			IF (GVL.A_RunStep <= GVL.A_LengthStep)
			   AND F_IsMotionCmd(
					GVL_1.Step_Cr_A[GVL.A_RunStep].Cmd
			   )
			THEN
	
				//----------------------------------------
				// Đồng bộ step tiếp theo cần Push
				//----------------------------------------
// 				GVL.A_PipelineNextPushStep :=
// 					GVL.A_RunStep;
				GVL.A_RunState := 100;
				IF (GVL.A_RunMode = 1) THEN
					GVL.A_StepHold := TRUE;
				END_IF;
				
	
			ELSE
	
				// Gặp END_WHILE hoặc logic khác
				GVL.A_RunState := 130;
	
			END_IF;
	
		END_IF;
		



    130: // WAIT ALL MOTION CLEAR BEFORE LOGIC

		//--------------------------------------------------------
		// Chờ queue và toàn bộ slot motion thực sự sạch
		//--------------------------------------------------------
		IF (GVL.A_MotionCount <= 0)
		   AND (GVL.A_ActiveMotionCount <= 0)
		   AND NOT GVL.A_MotionManagerBusy
		THEN
			//----------------------------------------------------
			// Reset trạng thái phiên pipeline vừa kết thúc
			//----------------------------------------------------
			GVL.A_PipelineActive := FALSE;
// 			GVL.A_PipelineNextPushStep := 0;
// 	
// 			GVL.A_PushMotionReq := FALSE;
// 			GVL.A_PushMotionDone := FALSE;
// 			GVL.A_PushMotionError := FALSE;
// 	
// 			//----------------------------------------------------
// 			// Xóa phản hồi completion của chuỗi motion vừa chạy
// 			//----------------------------------------------------
// 			GVL.A_MotionDonePulse := FALSE;
// 			GVL.A_MotionDoneStep := 0;
// 	
// 			GVL.A_MotionErrorPulse := FALSE;
// 			GVL.A_MotionErrorStep := 0;
// 			GVL.A_MotionErrorCode := 0;
	
			//----------------------------------------------------
			// Quay lại READ STEP để chạy lệnh logic:
			// END_WHILE, IF, WAIT, END...
			//----------------------------------------------------
			GVL.A_RunState := 0;
		END_IF;
		
	140: // WAIT MOTION CLEAR BEFORE WHILE RESTART

		//--------------------------------------------------------
		// Chờ toàn bộ motion của vòng hiện tại hoàn thành
		//--------------------------------------------------------
		IF (GVL.A_MotionCount <= 0)
		   AND (GVL.A_ActiveMotionCount <= 0)
		   AND NOT GVL.A_MotionManagerBusy
		THEN
			//----------------------------------------------------
			// Hạ request của pipeline
			//----------------------------------------------------
			GVL.A_PushMotionReq := FALSE;
			GVL.A_PipelineActive := FALSE;
	
			//----------------------------------------------------
			// Sang bước reset handshake
			//----------------------------------------------------
			MotionCycleResetScan := 0;
			GVL.A_RunState := 141;
		END_IF;
		
	141: // RESET MOTION PIPELINE BEFORE NEXT WHILE LOOP

		CASE MotionCycleResetScan OF
	
			0:
				//------------------------------------------------
				// Scan thứ nhất: xóa các tín hiệu phiên cũ
				//------------------------------------------------
				GVL.A_PushMotionReq := FALSE;
				GVL.A_PushMotionDone := FALSE;
				GVL.A_PushMotionError := FALSE;
	
				GVL.A_PipelineActive := FALSE;
				GVL.A_PipelineNextPushStep := 0;
	
				GVL.A_MotionDonePulse := FALSE;
				GVL.A_MotionDoneStep := 0;
	
				GVL.A_MotionErrorPulse := FALSE;
				GVL.A_MotionErrorStep := 0;
				GVL.A_MotionErrorCode := 0;
	
				MotionCycleResetScan := 1;
	
	
			1:
				//------------------------------------------------
				// Scan thứ hai:
				// fbPushMotion đã được gọi với Execute=FALSE.
				// Motion FB đã được gọi với Start=FALSE.
				//------------------------------------------------
				IF NOT GVL.A_PushMotionReq
				   AND (GVL.A_MotionCount <= 0)
				   AND (GVL.A_ActiveMotionCount <= 0)
				   AND NOT GVL.A_MotionManagerBusy
				THEN
					MotionCycleResetScan := 0;
	
					//--------------------------------------------
					// Bây giờ mới quay lại WHILE
					//--------------------------------------------
					GVL.A_RunStep := WhileReturnStep;
					GVL.A_RunState := 0;
				END_IF;
	
		END_CASE;
	
    900: // ERROR
        GVL.A_RunBusy := FALSE;
        GVL.A_PushMotionReq := FALSE;
        GVL.A_PipelineActive := FALSE;

END_CASE;


//====================================================
// FB Push Motion Queue phải gọi mỗi scan
//====================================================
fbPushMotion(
    Execute := GVL.A_PushMotionReq,
    Item := GVL.A_PushMotionItem
);

GVL.A_PushMotionDone  := fbPushMotion.Done;
GVL.A_PushMotionError := fbPushMotion.Error;
END_ACTION

ACTION PRG_A_MotionManager:
//====================================================
// PRG_A_MotionManager
// Controlled Pipeline Motion Manager
// - Chạy nền liên tục.
// - Có queue và slot rảnh thì Pop motion vào slot.
// - Slot Accepted thì hạ Start để FB Motion chạy tiếp.
// - Slot Done thì báo về Interpreter bằng A_MotionDonePulse.
// - Slot Error thì báo lỗi đúng SourceStep.
//====================================================


//====================================================
// ABORT REQUEST
// Ưu tiên cao nhất trong MotionManager
// Dùng khi Stop / Alarm / Reset
//====================================================
IF GVL.A_MotionAbortReq OR GVL.X[7] THEN

    PopReq := FALSE;

    GVL.A_MotionHead := 1;
    GVL.A_MotionTail := 1;
    GVL.A_MotionCount := 0;
	GVL.A_PipelineUsedCount := 0;
    FOR i := 1 TO 3 DO
        GVL.A_MoveSlotStart[i] := FALSE;
        GVL.A_MoveSlotBusy[i] := FALSE;

        GVL.A_MoveSlotAccepted[i] := FALSE;
        GVL.A_MoveSlotDone[i] := FALSE;
        GVL.A_MoveSlotError[i] := FALSE;
        GVL.A_MoveSlotErrorID[i] := 0;
		GVL.A_MoveSlotReleasePending[i] := FALSE;
        GVL.A_MoveSlotCmd[i] := E_RobotCmd.CMD_NOP;
		
    END_FOR;

    GVL.A_ActiveMotionCount := 0;

    GVL.A_MotionManagerBusy := FALSE;
    GVL.A_MotionManagerDone := FALSE;
    GVL.A_MotionManagerError := FALSE;
    GVL.A_MotionManagerState := 0;

    GVL.A_MotionDonePulse := FALSE;
    GVL.A_MotionErrorPulse := FALSE;

    GVL.A_MotionAbortReq := FALSE;
    GVL.A_MotionAbortDone := TRUE;

ELSE

	// Luôn gọi FB MoveP/L/C mỗi scan
	
	CASE GVL.A_MotionManagerState OF
	
		0: // IDLE / READY
	
			GVL.A_MotionManagerDone := FALSE;
	
			// Nếu có motion trong queue và còn slot rảnh thì lấy ra chạy
			IF (GVL.A_MotionCount > 0) AND (F_GetFreeMoveSlot() > 0) THEN
				GVL.A_MotionManagerBusy := TRUE;
				PopReq := TRUE;
	
				GVL.A_MotionManagerState := 10;
	
			ELSE
				// Không còn queue và không còn slot active
				IF GVL.A_ActiveMotionCount <= 0 THEN
					GVL.A_MotionManagerBusy := FALSE;
				END_IF;
			END_IF;
	
	
		10: // WAIT POP DONE
	
			IF fbPop.Done THEN
				PopReq := FALSE;
	
				item_PRG_A_MotionManager := fbPop.Item;
				freeSlot := F_GetFreeMoveSlot();
	
				IF freeSlot > 0 THEN
	
					// Gán item vào slot rảnh
					GVL.A_MoveSlotItem[freeSlot] := item_PRG_A_MotionManager;
					GVL.A_MoveSlotCmd[freeSlot]  := item_PRG_A_MotionManager.Cmd;
	
					// Reset trạng thái slot trước khi Start
					GVL.A_MoveSlotBusy[freeSlot]     := TRUE;
					GVL.A_MoveSlotStart[freeSlot]    := TRUE;
					GVL.A_MoveSlotAccepted[freeSlot] := FALSE;
					GVL.A_MoveSlotDone[freeSlot]     := FALSE;
					GVL.A_MoveSlotError[freeSlot]    := FALSE;
					
					GVL.A_MoveSlotErrorID[freeSlot] := 0;

					GVL.A_MoveSlotReleasePending[freeSlot] := FALSE;
					
					// Ghi nhớ chính xác slot vừa cấp
   					WaitAcceptSlot := freeSlot;
	
					// Tăng số motion đang active
					//GVL.A_ActiveMotionCount := GVL.A_ActiveMotionCount + 1;
	
					GVL.A_MotionManagerState := 20;
	
				ELSE
					// Trường hợp hiếm: vừa Pop xong nhưng slot không còn rảnh
					GVL.A_MotionManagerState := 30;
				END_IF;
			END_IF;
	
			IF fbPop.Empty THEN
				PopReq := FALSE;
				GVL.A_MotionManagerState := 30;
			END_IF;
	
	
		20: // WAIT COMMAND ACCEPTED
			
		//--------------------------------------------------------
			// Chỉ chờ đúng slot vừa được State 10 cấp lệnh
			//--------------------------------------------------------
			IF (WaitAcceptSlot >= 1)
			   AND (WaitAcceptSlot <= 3)
			THEN
		
				//----------------------------------------------------
				// Slot vẫn phải thuộc quyền sở hữu của Manager
				//----------------------------------------------------
				IF GVL.A_MoveSlotBusy[WaitAcceptSlot] THEN
		
					//------------------------------------------------
					// Lệnh đã được FB Move nhận
					//------------------------------------------------
					IF GVL.A_MoveSlotAccepted[WaitAcceptSlot] THEN
		
						GVL.A_MoveSlotStart[WaitAcceptSlot] := FALSE;
		
						// Đã hoàn thành handshake Accepted
						WaitAcceptSlot := 0;
		
						//--------------------------------------------
						// PipelineLength = 1:
						// Không Pop thêm khi còn motion đang chạy.
						// Sang State 30 chờ motion hoàn thành.
						//--------------------------------------------
						GVL.A_MotionManagerState := 30;
		
		
					ELSIF GVL.A_MoveSlotError[WaitAcceptSlot] THEN
		
						GVL.A_MotionManagerError := TRUE;
		
						GVL.A_MotionErrorPulse := TRUE;
						GVL.A_MotionErrorStep :=
							GVL.A_MoveSlotItem[WaitAcceptSlot].SourceStep;
		
						GVL.A_MotionErrorCode :=
							GVL.A_MoveSlotErrorID[WaitAcceptSlot];
		
						WaitAcceptSlot := 0;
		
						GVL.A_MotionManagerState := 900;
		
					END_IF;
		
				END_IF;
		
			ELSE
		
				//----------------------------------------------------
				// Không có slot nào đang chờ Accepted.
				// Đây là trạng thái bất thường, quay về quản lý queue.
				//----------------------------------------------------
				GVL.A_MotionManagerState := 30;
		
			END_IF;
	
		30: // WAIT / CONTINUE PIPELINE
	
			// Nếu sau đó Interpreter push thêm queue và có slot rảnh thì tiếp tục chạy
			IF (GVL.A_MotionCount > 0) AND (F_GetFreeMoveSlot() > 0) THEN
				GVL.A_MotionManagerBusy := TRUE;
				PopReq := TRUE;
				GVL.A_MotionManagerState := 10;
	
			// Nếu không còn queue và không còn motion active thì MotionManager rảnh
			ELSIF (GVL.A_MotionCount <= 0) AND (GVL.A_ActiveMotionCount <= 0) THEN
				GVL.A_MotionManagerBusy := FALSE;
				GVL.A_MotionManagerDone := TRUE;
				GVL.A_MotionManagerState := 0;
			END_IF;
	
	
		900: // ERROR
	
			PopReq := FALSE;
	
			// Dừng cấp thêm motion mới
			FOR i := 1 TO 3 DO
				GVL.A_MoveSlotStart[i] := FALSE;
			END_FOR;
	
			GVL.A_MotionManagerBusy := FALSE;
			GVL.A_MotionManagerError := TRUE;
	
			GVL.A_MotionManagerState := 0;
	
	END_CASE;
END_IF;
//====================================================
// Gọi FB Pop mỗi scan
//====================================================
fbPop(
    Execute := PopReq
);



//============================================================
// CALL MOTION SLOT FB
// Tất cả FB phải được gọi liên tục mỗi scan.
//
// Khi slot không sử dụng hoặc không đúng loại lệnh:
// Start của FB tương ứng phải bằng FALSE.
// Nhờ vậy LastStart và State bên trong FB được cập nhật đúng.
//============================================================

FOR i := 1 TO 3 DO

    //--------------------------------------------------------
    // Chuẩn bị tọa độ
    //--------------------------------------------------------
    IF GVL.A_MoveSlotBusy[i] THEN

        CASE GVL.A_MoveSlotCmd[i] OF

            E_RobotCmd.CMD_MovP,
            E_RobotCmd.CMD_MovL:

//                 SlotPos[i] :=
//                     F_GetPointSMC_A(
//                         GVL.A_MoveSlotItem[i].PointNo
//                     );
				IF GVL.A_MoveSlotItem[i].UseDirectPosition THEN
					SlotPos[i].c.X := GVL.A_MoveSlotItem[i].DirectPosition.X;
					SlotPos[i].c.Y := GVL.A_MoveSlotItem[i].DirectPosition.Y;
					SlotPos[i].c.Z := GVL.A_MoveSlotItem[i].DirectPosition.Z;
					SlotPos[i].c.A := GVL.A_MoveSlotItem[i].DirectPosition.A;
				ELSE
					SlotPos[i] := F_GetPointSMC_A(GVL.A_MoveSlotItem[i].PointNo);
				END_IF;



            E_RobotCmd.CMD_MovC:

                SlotMidPos[i] :=
                    F_GetPointSMC_A(
                        GVL.A_MoveSlotItem[i].MidPointNo
                    );

                SlotEndPos[i] :=
                    F_GetPointSMC_A(
                        GVL.A_MoveSlotItem[i].EndPointNo
                    );

        END_CASE;

    END_IF;


    //--------------------------------------------------------
    // MoveP
    // Luôn gọi mỗi scan
    //--------------------------------------------------------
    fbMoveP[i](
        Start :=
            GVL.A_MoveSlotBusy[i]
            AND
            (GVL.A_MoveSlotCmd[i] = E_RobotCmd.CMD_MovP)
            AND
            GVL.A_MoveSlotStart[i],
		Release := GVL.A_MoveSlotReleasePending[i],
        AxisGroup := SCARA_A,
        Item := GVL.A_MoveSlotItem[i],
        PositionIn := SlotPos[i],
        //CoordSystem := GVL.RB_A.COORD
		CoordSystem := SEL(
			GVL.A_MoveSlotItem[i].UseDirectPosition,
			//GVL.RB_A.COORD,
			SMC_COORD_SYSTEM.MCS,
			GVL.A_MoveSlotItem[i].DirectCoordSystem)

    );


    //--------------------------------------------------------
    // MoveL
    // Luôn gọi mỗi scan
    //--------------------------------------------------------
    fbMoveL[i](
        Start :=
            GVL.A_MoveSlotBusy[i]
            AND
            (GVL.A_MoveSlotCmd[i] = E_RobotCmd.CMD_MovL)
            AND
            GVL.A_MoveSlotStart[i],

        AxisGroup := SCARA_A,
        Item := GVL.A_MoveSlotItem[i],
        PositionIn := SlotPos[i],
        //CoordSystem := GVL.RB_A.COORD
		CoordSystem := SEL(
			GVL.A_MoveSlotItem[i].UseDirectPosition,
			//GVL.RB_A.COORD,
			SMC_COORD_SYSTEM.MCS,
			GVL.A_MoveSlotItem[i].DirectCoordSystem)

    );


    //--------------------------------------------------------
    // MoveC
    // Luôn gọi mỗi scan
    //--------------------------------------------------------
    fbMoveC[i](
        Start :=
            GVL.A_MoveSlotBusy[i]
            AND
            (GVL.A_MoveSlotCmd[i] = E_RobotCmd.CMD_MovC)
            AND
            GVL.A_MoveSlotStart[i],

        AxisGroup := SCARA_A,
        Item := GVL.A_MoveSlotItem[i],
        MidPosition := SlotMidPos[i],
        EndPosition := SlotEndPos[i],
        //CoordSystem := GVL.RB_A.COORD
		CoordSystem := SMC_COORD_SYSTEM.MCS
    );


	



    //--------------------------------------------------------
    // Chọn trạng thái trả về theo loại lệnh của slot
    //--------------------------------------------------------
    IF GVL.A_MoveSlotBusy[i] THEN

        CASE GVL.A_MoveSlotCmd[i] OF

            //================================================
            // MOVP
            //================================================
            E_RobotCmd.CMD_MovP:

                GVL.A_MoveSlotAccepted[i] :=
                    fbMoveP[i].Accepted;

                GVL.A_MoveSlotDone[i] :=
                    fbMoveP[i].Done;

                GVL.A_MoveSlotError[i] :=
                    fbMoveP[i].Error;

                GVL.A_MoveSlotErrorID[i] :=
                    fbMoveP[i].ErrorID_Custom;


            //================================================
            // MOVL
            //================================================
            E_RobotCmd.CMD_MovL:

                GVL.A_MoveSlotAccepted[i] :=
                    fbMoveL[i].Accepted;

                GVL.A_MoveSlotDone[i] :=
                    fbMoveL[i].Done;

                GVL.A_MoveSlotError[i] :=
                    fbMoveL[i].Error;

                GVL.A_MoveSlotErrorID[i] :=
                    fbMoveL[i].ErrorID_Custom;


            //================================================
            // MOVC
            //================================================
            E_RobotCmd.CMD_MovC:

                GVL.A_MoveSlotAccepted[i] :=
                    fbMoveC[i].Accepted;

                GVL.A_MoveSlotDone[i] :=
                    fbMoveC[i].Done;

                GVL.A_MoveSlotError[i] :=
                    fbMoveC[i].Error;

                GVL.A_MoveSlotErrorID[i] :=
                    fbMoveC[i].ErrorID_Custom;

        END_CASE;

    END_IF;

END_FOR;


//------------------------------------------------------------
// GLOBAL MOTION ERROR MONITOR
//
// Kiểm tra tất cả Move Slot mỗi scan.
// Giữ nguyên cơ chế MotionErrorPulse cũ để báo Interpreter.
//------------------------------------------------------------
IF NOT GVL.A_MotionErrorPulse THEN

    FOR i := 1 TO 3 DO

        IF GVL.A_MoveSlotBusy[i] AND GVL.A_MoveSlotError[i]
        THEN

            //--------------------------------------------
            // MotionManager có lỗi
            //--------------------------------------------
            GVL.A_MotionManagerError := TRUE;

            //--------------------------------------------
            // Xung báo Interpreter
            //--------------------------------------------
            GVL.A_MotionErrorPulse := TRUE;

            //--------------------------------------------
            // Step gây lỗi
            //--------------------------------------------
            GVL.A_MotionErrorStep := GVL.A_MoveSlotItem[i].SourceStep;

            //--------------------------------------------
            // Error Code của FB
            //--------------------------------------------
            GVL.A_MotionErrorCode := GVL.A_MoveSlotErrorID[i];

            //--------------------------------------------
            // Có thể lưu thêm Slot để debug
            //--------------------------------------------
            GVL.A_MotionErrorSlot := i;

            //--------------------------------------------
            // Manager chuyển ERROR
            //--------------------------------------------
            GVL.A_MotionManagerState := 900;

            EXIT;

        END_IF;

    END_FOR;

END_IF;

// RELEASE SLOT WHEN DONE
FOR i := 1 TO 3 DO

    IF GVL.A_MoveSlotBusy[i]
       AND GVL.A_MoveSlotDone[i]
    THEN

        // Báo Interpreter
        GVL.A_MotionDoneStep :=
            GVL.A_MoveSlotItem[i].SourceStep;

        GVL.A_MotionDonePulse := TRUE;

        // Release slot
        GVL.A_MoveSlotStart[i] := FALSE;
        GVL.A_MoveSlotBusy[i] := FALSE;
        GVL.A_MoveSlotAccepted[i] := FALSE;
        GVL.A_MoveSlotDone[i] := FALSE;
        GVL.A_MoveSlotError[i] := FALSE;
        GVL.A_MoveSlotErrorID[i] := 0;

        GVL.A_MoveSlotCmd[i] :=
            E_RobotCmd.CMD_NOP;
		GVL.A_MoveSlotReleasePending[i] := TRUE; // Set release = TRUE
		
		//------------------------------------------------
		// Motion đã thực sự rời pipeline
		//------------------------------------------------
		IF GVL.A_PipelineUsedCount > 0 THEN
			GVL.A_PipelineUsedCount :=
				GVL.A_PipelineUsedCount - 1;
		END_IF;
	
    END_IF;
END_FOR;

//============================================================
// RECALCULATE ACTIVE MOTION COUNT
//
// A_ActiveMotionCount luôn phản ánh đúng số slot Busy,
// không phụ thuộc việc cộng/trừ có bị bỏ sót hay không.
//============================================================
ActiveCountCalc := 0;

FOR i := 1 TO 3 DO

    IF GVL.A_MoveSlotBusy[i] THEN
        ActiveCountCalc := ActiveCountCalc + 1;
    END_IF;

END_FOR;

GVL.A_ActiveMotionCount := ActiveCountCalc;




//====================================================
// FINALIZE MOTION MANAGER
// Chỉ kết thúc khi Manager đã vào trạng thái WAIT
// Không được reset State 10/20 khi vừa Pop lệnh.
//====================================================
IF (GVL.A_MotionManagerState = 30)
   AND (GVL.A_MotionCount <= 0)
   AND (GVL.A_ActiveMotionCount <= 0)
THEN

    GVL.A_MotionManagerBusy := FALSE;
    GVL.A_MotionManagerDone := TRUE;
    GVL.A_MotionManagerState := 0;

END_IF;
END_ACTION

ACTION Main_Base_Program_RB_B:
//=============================================================================
// REPLACE ACTION: Main_Base_Program_RB_B
// SOURCE: current Main_Base_Program_RB_A in PG_MAR_V3_1707_10(4).xml
// METHOD: strict A -> B mirror for robot-specific runtime.
// IMPORTANT: replace the ENTIRE existing Main_Base_Program_RB_B body.
//=============================================================================

//====================================================
// PRG_B_Interpreter
// Controlled Pipeline:
// - Motion được nạp trước tối đa A_PipelineDepth lệnh.
// - A_RunStep chỉ tăng khi step hiện tại Done thật.
// - Gặp lệnh logic thì chờ Motion Queue + Slot sạch.
//====================================================



//====================================================
// STOP COMMAND
//====================================================
IF GVL.B_RunStop OR GVL.X[7] THEN

    // Dừng Interpreter
    GVL.B_RunEnable := FALSE;
    GVL.B_RunBusy := FALSE;
    GVL.B_RunDone := FALSE;
    GVL.B_RunPause := FALSE;
    GVL.B_RunState := 0;
    // GVL.B_RunStop := FALSE;

    // Dừng pipeline
    GVL.B_PipelineActive := FALSE;
    GVL.B_PushMotionReq := FALSE;
    GVL.B_PushMotionDone := FALSE;
    GVL.B_PushMotionError := FALSE;
	// 1707
	//------------------------------------------------
    // Reset bộ nhớ cạnh của FB Push
    //------------------------------------------------
    fbPushMotion_B(
        Execute := FALSE,
        Item := GVL.B_PushMotionItem
    );

    // Yêu cầu MotionManager abort toàn bộ motion pipeline
    GVL.B_MotionAbortReq := TRUE;
	
	// Dừng command Tracking đang chạy.
	IF GVL.B_StepActive THEN
		GVL.g_stMultiTrackCommandB.Abort := TRUE;
		GVL.g_stMultiTrackCommandB.Execute := FALSE;
	
		GVL.B_StepActive := FALSE;
		udiTrackCommandIDB := 0;
	END_IF;
	
	// Hủy Tool command từ Interpreter.
	GVL.g_stInterpreterToolCommandB.Execute := FALSE;
	GVL.g_stInterpreterToolCommandB.Abort := TRUE;
	
	udiToolReleaseCommandIDB := 0;
	// GVL.B_StepActive := FALSE;
	//GVL.g_axDORequestToolB[4] := FALSE;
	
	//xVisionAlignStartB := FALSE;
	// Hủy Vision Request khi Stop/Disable Robot B.

    //=============================================================================
	// ABORT VISION REQUEST - ROBOT B
	//-----------------------------------------------------------------------------
	// Khi Robot Stop, Robot không phát Request mới và hạ Execute hiện tại.
	// Vision Manager sẽ thực hiện phần reset handshake phía Manager.
	//=============================================================================
	GVL.g_stVisionAlignRequestB.Execute := FALSE;
	xVisionStepActiveB := FALSE;

    RETURN;
END_IF;


//====================================================
// NOT ENABLE
//====================================================
IF NOT GVL.B_RunEnable THEN
    GVL.B_RunBusy := FALSE;
    GVL.B_RunState := 0;
    GVL.B_PushMotionReq := FALSE;
    GVL.B_PipelineActive := FALSE;
	GVL.B_RunAlarm := FALSE;
	GVL.B_RunStep := 1;
	
	GVL.g_stMultiTrackCommandB.Execute := FALSE;
	GVL.g_stMultiTrackCommandB.Abort := FALSE;
	GVL.g_stMultiTrackCommandB.Reset := FALSE;
	
	GVL.B_StepActive := FALSE;
	udiTrackCommandIDB := 0;
	
	GVL.g_stInterpreterToolCommandB.Execute := FALSE;
	GVL.g_stInterpreterToolCommandB.Abort := FALSE;
	GVL.g_stInterpreterToolCommandB.Reset := FALSE;
	
	udiToolReleaseCommandIDB := 0;
	
	// Reset command Vision của Interpreter.
	//xVisionAlignStartB := FALSE;
// 	uiVisionCameraIDB := 1;
// 	uiVisionJobIDB := 1;

	// Hủy Vision Request khi Stop/Disable Robot B.

    GVL.g_stVisionAlignRequestB.Execute := FALSE;   // Hạ Request để Manager kết thúc handshake.

    xVisionStepActiveB := FALSE;                    // Xóa ownership command Vision Robot B.

    uiVisionCameraIDB := 1;                         // Reset CameraID mặc định nếu cần.

    uiVisionJobIDB := 1;                            // Reset JobID mặc định nếu cần.

    iVisionResultVarB := 0;                         // Reset index biến kết quả.
	
	GVL.B_VisionDone := FALSE;
	GVL.B_VisionOK := FALSE;
	GVL.B_VisionError := FALSE;

    RETURN;
END_IF;


//====================================================
// PAUSE
// Pause chỉ dừng Interpreter, không reset Motion đang chạy
//====================================================
IF GVL.B_RunPause THEN
    GVL.B_RunBusy := TRUE;
    RETURN;
END_IF;


//====================================================
// ALARM
//====================================================
IF GVL.B_RunAlarm THEN
    GVL.B_RunBusy := FALSE;
    GVL.B_PushMotionReq := FALSE;
    GVL.B_PipelineActive := FALSE;

    // Khi lỗi thì yêu cầu MotionManager ngừng cấp lệnh mới
    GVL.B_MotionAbortReq := TRUE;

    RETURN;
END_IF;


//====================================================
// RUNNING
//====================================================
GVL.B_RunBusy := TRUE;


//====================================================
// CHECK STEP RANGE
//====================================================
IF GVL.B_RunStep < 1 THEN
    GVL.B_RunStep := 1;
END_IF;

IF GVL.B_RunStep > GVL.B_LengthStep THEN
    GVL.B_RunEnable := FALSE;
    GVL.B_RunBusy := FALSE;
    GVL.B_RunDone := TRUE;
    GVL.B_RunState := 0;
    GVL.B_PipelineActive := FALSE;
    GVL.B_PushMotionReq := FALSE;
	GVL.B_RunStep := 1;
    RETURN;
END_IF;


//====================================================
// STEP RUN EDGE
// Bắt xung nút chạy từng bước từ HMI
//====================================================
GVL.B_StepRunEdge := GVL.B_StepRunReq AND NOT GVL.B_LastStepRunReq;
GVL.B_LastStepRunReq := GVL.B_StepRunReq;


//====================================================
// STEP HOLD
// Nếu đang ở chế độ Step và đang Hold
// thì chỉ chạy tiếp khi có xung StepRun
//====================================================
IF GVL.B_RunMode = 1 THEN

    IF GVL.B_StepHold THEN

        IF GVL.B_StepRunEdge THEN
            // Cho phép chạy 1 step tiếp theo
            GVL.B_StepHold := FALSE;
        ELSE
            // Chưa bấm Step thì đứng yên
            GVL.B_RunBusy := TRUE;
            RETURN;
        END_IF;

    END_IF;

END_IF;


CASE GVL.B_RunState OF

    0: // READ STEP

        step_PRG_B_Interpreter := GVL_1.Step_Cr_B[GVL.B_RunStep];

        IF F_IsMotionCmd(step_PRG_B_Interpreter.Cmd) THEN

            // Bắt đầu pipeline tại step hiện tại
            GVL.B_PipelineActive := TRUE;

            // Step tiếp theo cần push vào motion queue
            GVL.B_PipelineNextPushStep := GVL.B_RunStep;

            GVL.B_RunState := 100;

        ELSE

            // Lệnh logic chỉ được chạy khi toàn bộ motion đã sạch
            IF (GVL.B_MotionCount <= 0) AND (GVL.B_ActiveMotionCount <= 0) THEN
                GVL.B_RunState := 10;
            ELSE
                GVL.B_RunState := 130;
            END_IF;

        END_IF;


    10: // EXECUTE LOGIC COMMAND

        step_PRG_B_Interpreter := GVL_1.Step_Cr_B[GVL.B_RunStep];

        CASE step_PRG_B_Interpreter.Cmd OF

            E_RobotCmd.CMD_NOP:
                GVL.B_RunStep := GVL.B_RunStep + 1;
                GVL.B_RunState := 0;


            E_RobotCmd.CMD_Set_Speed:
                // P1 = Speed, P2 = Acc, P3 = Dec, P4 = Jerk
                GVL.B_CurrentMotionParam.Speed := INT_TO_LREAL(step_PRG_B_Interpreter.P1);
                GVL_1.DATA_RB_B.MOTION_ACC  := INT_TO_LREAL(step_PRG_B_Interpreter.P2);
                GVL_1.DATA_RB_B.MOTION_DEC  := DINT_TO_LREAL(step_PRG_B_Interpreter.P3);
                GVL_1.DATA_RB_B.MOTION_JERK := INT_TO_LREAL(step_PRG_B_Interpreter.P4);

                GVL.B_RunStep := GVL.B_RunStep + 1;
                GVL.B_RunState := 0;
				// Nếu đang Step Mode thì dừng chờ sau khi chạy xong 1 lệnh
				IF GVL.B_RunMode = 1 THEN
					GVL.B_StepHold := TRUE;
				END_IF;

            E_RobotCmd.CMD_Set_Fac_Speed:
                // P1 = VelFac %, P2 = AccFac %, P4 = JerkFac %
                GVL_1.DATA_RB_B.Fac_Vel  := INT_TO_LREAL(step_PRG_B_Interpreter.P1) / 100.0;
                GVL_1.DATA_RB_B.Fac_Acc  := INT_TO_LREAL(step_PRG_B_Interpreter.P2) / 100.0;
                GVL_1.DATA_RB_B.Fac_Jerk := INT_TO_LREAL(step_PRG_B_Interpreter.P4) / 100.0;

                IF GVL_1.DATA_RB_B.Fac_Vel <= 0.0 THEN GVL_1.DATA_RB_B.Fac_Vel := 0.1; END_IF;
                IF GVL_1.DATA_RB_B.Fac_Acc <= 0.0 THEN GVL_1.DATA_RB_B.Fac_Acc := 0.1; END_IF;
                IF GVL_1.DATA_RB_B.Fac_Jerk <= 0.0 THEN GVL_1.DATA_RB_B.Fac_Jerk := 0.1; END_IF;

                GVL.B_RunStep := GVL.B_RunStep + 1;
                GVL.B_RunState := 0;
				
				// Nếu đang Step Mode thì dừng chờ sau khi chạy xong 1 lệnh
				IF GVL.B_RunMode = 1 THEN
					GVL.B_StepHold := TRUE;
				END_IF;

			// DIGITAL OUTPUT
            E_RobotCmd.CMD_DO_ON:
				// P1 = Output No;
				GVL.Y[step_PRG_B_Interpreter.P1] := TRUE;

                GVL.B_RunStep := GVL.B_RunStep + 1;
                GVL.B_RunState := 0;
				
				// Nếu đang Step Mode thì dừng chờ sau khi chạy xong 1 lệnh
				IF GVL.B_RunMode = 1 THEN
					GVL.B_StepHold := TRUE;
				END_IF;


            E_RobotCmd.CMD_DO_OFF:
                // P1 = Output No;
				GVL.Y[step_PRG_B_Interpreter.P1] := FALSE;

                GVL.B_RunStep := GVL.B_RunStep + 1;
                GVL.B_RunState := 0;
				
				// Nếu đang Step Mode thì dừng chờ sau khi chạy xong 1 lệnh
				IF GVL.B_RunMode = 1 THEN
					GVL.B_StepHold := TRUE;
				END_IF;

			E_RobotCmd.CMD_DO_TOGGLE:
				// P1 = Output No;
				GVL.Y[step_PRG_B_Interpreter.P1] := NOT GVL.Y[step_PRG_B_Interpreter.P1];
				GVL.B_RunStep := GVL.B_RunStep + 1;
				GVL.B_RunState := 0;
				
				// Nếu đang Step Mode thì dừng chờ sau khi chạy xong 1 lệnh
				IF GVL.B_RunMode = 1 THEN
					GVL.B_StepHold := TRUE;
				END_IF;

			 //================================================
			// WAIT
			//================================================
			E_RobotCmd.CMD_WAIT_IN:
				// P1=Input No, P2=Expected 0/1
				IF GVL.X[step_PRG_B_Interpreter.P1] = (step_PRG_B_Interpreter.P2 <> 0) THEN
					GVL.B_RunStep := GVL.B_RunStep + 1;
					GVL.B_RunState := 0;
					// Nếu đang Step Mode thì dừng chờ sau khi chạy xong 1 lệnh
					IF GVL.B_RunMode = 1 THEN
						GVL.B_StepHold := TRUE;
					END_IF;
				END_IF;
			
			E_RobotCmd.CMD_WAIT:
				// P1=Condition No
				IF F_EvalCondition_B(step_PRG_B_Interpreter.P1) THEN
					GVL.B_RunStep := GVL.B_RunStep + 1;
					GVL.B_RunState := 0;
					// Nếu đang Step Mode thì dừng chờ sau khi chạy xong 1 lệnh
					IF GVL.B_RunMode = 1 THEN
						GVL.B_StepHold := TRUE;
					END_IF;
				END_IF;
            
            E_RobotCmd.CMD_Delay:
                // P1 = thời gian delay ms
                tRunDelay_B(IN := TRUE, PT := INT_TO_TIME(step_PRG_B_Interpreter.P1));

                IF tRunDelay_B.Q THEN
                    tRunDelay_B(IN := FALSE);
                    GVL.B_RunStep := GVL.B_RunStep + 1;
                    GVL.B_RunState := 0;
					// Nếu đang Step Mode thì dừng chờ sau khi chạy xong 1 lệnh
					IF GVL.B_RunMode = 1 THEN
						GVL.B_StepHold := TRUE;
					END_IF;
                END_IF;

			//================================================
			// TIMER
			//================================================
			E_RobotCmd.CMD_Timer_Start:
				// P1=Timer No, P2=Time ms
				GVL.B_TimerPT[step_PRG_B_Interpreter.P1] := DINT_TO_TIME(step_PRG_B_Interpreter.P2);
				GVL.B_TimerStart[step_PRG_B_Interpreter.P1] := TRUE;
				GVL.B_TimerDone[step_PRG_B_Interpreter.P1] := FALSE;
	
				GVL.B_RunStep := GVL.B_RunStep + 1;
				GVL.B_RunState := 0;
				
				// Nếu đang Step Mode thì dừng chờ sau khi chạy xong 1 lệnh
				IF GVL.B_RunMode = 1 THEN
					GVL.B_StepHold := TRUE;
				END_IF;
	
	
			E_RobotCmd.CMD_Timer_Wait:
				// P1=Timer No
				IF GVL.B_TimerDone[step_PRG_B_Interpreter.P1] THEN
					GVL.B_TimerStart[step_PRG_B_Interpreter.P1] := FALSE;
					GVL.B_RunStep := GVL.B_RunStep + 1;
					GVL.B_RunState := 0;
					// Nếu đang Step Mode thì dừng chờ sau khi chạy xong 1 lệnh
					IF GVL.B_RunMode = 1 THEN
						GVL.B_StepHold := TRUE;
					END_IF;
				END_IF;
				
			//================================================
			// IF / ELSE
			//================================================
			E_RobotCmd.CMD_IF:
				// P1=Condition No
				IF F_EvalCondition_B(step_PRG_B_Interpreter.P1) THEN
					GVL.B_RunStep := GVL.B_RunStep + 1;
					// Nếu đang Step Mode thì dừng chờ sau khi chạy xong 1 lệnh
					IF GVL.B_RunMode = 1 THEN
						GVL.B_StepHold := TRUE;
					END_IF;
				ELSE
					GVL.B_RunStep := F_FindElseOrEndIf_B(GVL.B_RunStep);
					// Nếu đang Step Mode thì dừng chờ sau khi chạy xong 1 lệnh
					IF GVL.B_RunMode = 1 THEN
						GVL.B_StepHold := TRUE;
					END_IF;
				END_IF;
				GVL.B_RunState := 0;
	
	
			E_RobotCmd.CMD_IF_IN:
				// P1=Input No, P2=Expected 0/1
				IF GVL.X[step_PRG_B_Interpreter.P1] = (step_PRG_B_Interpreter.P2 <> 0) THEN
					GVL.B_RunStep := GVL.B_RunStep + 1;
					// Nếu đang Step Mode thì dừng chờ sau khi chạy xong 1 lệnh
					IF GVL.B_RunMode = 1 THEN
						GVL.B_StepHold := TRUE;
					END_IF;
				ELSE
					GVL.B_RunStep := F_FindElseOrEndIf_B(GVL.B_RunStep);
					// Nếu đang Step Mode thì dừng chờ sau khi chạy xong 1 lệnh
					IF GVL.B_RunMode = 1 THEN
						GVL.B_StepHold := TRUE;
					END_IF;
				END_IF;
				GVL.B_RunState := 0;
	
	
			E_RobotCmd.CMD_IF_VAR:
				// P1=Var No, P2=Operator, P3=SetValue
				IF F_CompareDINT_B(
					Actual := GVL.B_Var[step_PRG_B_Interpreter.P1],
					Operator := step_PRG_B_Interpreter.P2,
					SetValue := step_PRG_B_Interpreter.P3)
				THEN
					GVL.B_RunStep := GVL.B_RunStep + 1;
					// Nếu đang Step Mode thì dừng chờ sau khi chạy xong 1 lệnh
					IF GVL.B_RunMode = 1 THEN
						GVL.B_StepHold := TRUE;
					END_IF;
				ELSE
					GVL.B_RunStep := F_FindElseOrEndIf_B(GVL.B_RunStep);
					// Nếu đang Step Mode thì dừng chờ sau khi chạy xong 1 lệnh
					IF GVL.B_RunMode = 1 THEN
						GVL.B_StepHold := TRUE;
					END_IF;
				END_IF;
				GVL.B_RunState := 0;
	
	
			E_RobotCmd.CMD_IF_REG:
				// P1=Reg No, P2=Operator, P3=SetValue
				IF F_CompareDINT_B(
					Actual := GVL.B_Reg[step_PRG_B_Interpreter.P1],
					Operator := step_PRG_B_Interpreter.P2,
					SetValue := step_PRG_B_Interpreter.P3)
				THEN
					GVL.B_RunStep := GVL.B_RunStep + 1;
					// Nếu đang Step Mode thì dừng chờ sau khi chạy xong 1 lệnh
					IF GVL.B_RunMode = 1 THEN
						GVL.B_StepHold := TRUE;
					END_IF;
				ELSE
					GVL.B_RunStep := F_FindElseOrEndIf_B(GVL.B_RunStep);
					// Nếu đang Step Mode thì dừng chờ sau khi chạy xong 1 lệnh
					IF GVL.B_RunMode = 1 THEN
						GVL.B_StepHold := TRUE;
					END_IF;
				END_IF;
				GVL.B_RunState := 0;
	
	
			E_RobotCmd.CMD_ELSE:
				GVL.B_RunStep := F_FindEndIf_B(GVL.B_RunStep);
				GVL.B_RunState := 0;
				// Nếu đang Step Mode thì dừng chờ sau khi chạy xong 1 lệnh
				IF GVL.B_RunMode = 1 THEN
					GVL.B_StepHold := TRUE;
				END_IF;
	
			E_RobotCmd.CMD_END_IF:
				GVL.B_RunStep := GVL.B_RunStep + 1;
				GVL.B_RunState := 0;
				// Nếu đang Step Mode thì dừng chờ sau khi chạy xong 1 lệnh
				IF GVL.B_RunMode = 1 THEN
					GVL.B_StepHold := TRUE;
				END_IF;
			
			//================================================
			// JUMP / CALL / RETURN
			//================================================
			E_RobotCmd.CMD_JUMP:
				// P1=Target Step
				GVL.B_RunStep := step_PRG_B_Interpreter.P1;
				GVL.B_RunState := 0;
				// Nếu đang Step Mode thì dừng chờ sau khi chạy xong 1 lệnh
				IF GVL.B_RunMode = 1 THEN
					GVL.B_StepHold := TRUE;
				END_IF;
	
	
			E_RobotCmd.CMD_CALL:
				// P1=Target Step
				IF GVL.B_CallStackIndex < 20 THEN
					GVL.B_CallStackIndex := GVL.B_CallStackIndex + 1;
					GVL.B_CallStack[GVL.B_CallStackIndex] := GVL.B_RunStep + 1;
					GVL.B_RunStep := step_PRG_B_Interpreter.P1;
					GVL.B_RunState := 0;
				ELSE
					GVL.B_RunAlarm := TRUE;
					GVL.B_RunAlarmCode := 2101; // Call stack full
					GVL.B_RunErrorStep := GVL.B_RunStep;
					GVL.B_RunState := 900;
				END_IF;
	
	
			E_RobotCmd.CMD_RETURN:
				IF GVL.B_CallStackIndex > 0 THEN
					GVL.B_RunStep := GVL.B_CallStack[GVL.B_CallStackIndex];
					GVL.B_CallStackIndex := GVL.B_CallStackIndex - 1;
					GVL.B_RunState := 0;
				ELSE
					GVL.B_RunAlarm := TRUE;
					GVL.B_RunAlarmCode := 2102; // Return stack empty
					GVL.B_RunErrorStep := GVL.B_RunStep;
					GVL.B_RunState := 900;
				END_IF;
			
			//================================================
			// WHILE
			//================================================
			E_RobotCmd.CMD_WHILE:
				// P1=Condition No
				IF F_EvalCondition_B(step_PRG_B_Interpreter.P1) THEN
					GVL.B_RunStep := GVL.B_RunStep + 1;
					// Nếu đang Step Mode thì dừng chờ sau khi chạy xong 1 lệnh
					IF GVL.B_RunMode = 1 THEN
						GVL.B_StepHold := TRUE;
					END_IF;
				ELSE
					GVL.B_RunStep := F_FindEndWhile_B(GVL.B_RunStep);
					// Nếu đang Step Mode thì dừng chờ sau khi chạy xong 1 lệnh
					IF GVL.B_RunMode = 1 THEN
						GVL.B_StepHold := TRUE;
					END_IF;
				END_IF;
				GVL.B_RunState := 0;
	
	
			E_RobotCmd.CMD_WHILE_IN:
				// P1=Input No, P2=Expected 0/1
				IF GVL.X[step_PRG_B_Interpreter.P1] = (step_PRG_B_Interpreter.P2 <> 0) THEN
					GVL.B_RunStep := GVL.B_RunStep + 1;
					// Nếu đang Step Mode thì dừng chờ sau khi chạy xong 1 lệnh
					IF GVL.B_RunMode = 1 THEN
						GVL.B_StepHold := TRUE;
					END_IF;
				ELSE
					GVL.B_RunStep := F_FindEndWhile_B(GVL.B_RunStep);
					// Nếu đang Step Mode thì dừng chờ sau khi chạy xong 1 lệnh
					IF GVL.B_RunMode = 1 THEN
						GVL.B_StepHold := TRUE;
					END_IF;
				END_IF;
				GVL.B_RunState := 0;
	
	
			E_RobotCmd.CMD_WHILE_REG:
				// P1=Reg No, P2=Operator, P3=SetValue
				IF F_CompareDINT_B(
					Actual := GVL.B_Reg[step_PRG_B_Interpreter.P1],
					Operator := step_PRG_B_Interpreter.P2,
					SetValue := step_PRG_B_Interpreter.P3)
				THEN
					GVL.B_RunStep := GVL.B_RunStep + 1;
					// Nếu đang Step Mode thì dừng chờ sau khi chạy xong 1 lệnh
					IF GVL.B_RunMode = 1 THEN
						GVL.B_StepHold := TRUE;
					END_IF;
				ELSE
					GVL.B_RunStep := F_FindEndWhile_B(GVL.B_RunStep);
					// Nếu đang Step Mode thì dừng chờ sau khi chạy xong 1 lệnh
					IF GVL.B_RunMode = 1 THEN
						GVL.B_StepHold := TRUE;
					END_IF;
				END_IF;
				GVL.B_RunState := 0;
	
	
			E_RobotCmd.CMD_END_WHILE:
// 				GVL.B_RunStep := F_FindWhileStart_B(GVL.B_RunStep);
// 				GVL.B_RunState := 0;

				//--------------------------------------------------------
				// Lưu vị trí WHILE cần quay lại
				//--------------------------------------------------------
				WhileReturnStep_B :=
					F_FindWhileStart_B(GVL.B_RunStep);

				//--------------------------------------------------------
				// Không nhảy về WHILE ngay.
				// Trước tiên chờ pipeline của vòng hiện tại sạch.
				//--------------------------------------------------------
				GVL.B_RunState := 140;
				
				// Nếu đang Step Mode thì dừng chờ sau khi chạy xong 1 lệnh
				IF GVL.B_RunMode = 1 THEN
					GVL.B_StepHold := TRUE;
				END_IF;
			
// 			//================================================
// 			// VISION
// 			//================================================
// 			E_RobotCmd.CMD_VISION_TRIGGER:
// 				GVL.B_VisionTriggerReq := TRUE;
// 				GVL.B_RunStep := GVL.B_RunStep + 1;
// 				GVL.B_RunState := 0;
// 				// Nếu đang Step Mode thì dừng chờ sau khi chạy xong 1 lệnh
// 				IF GVL.B_RunMode = 1 THEN
// 					GVL.B_StepHold := TRUE;
// 				END_IF;

			E_RobotCmd.CMD_VISION_TRIGGER:
				//=========================================================================
				// VISION TRIGGER - ROBOT B
				//-------------------------------------------------------------------------
				// Command này thực hiện toàn bộ transaction:
				//
				// Robot B -> Vision Manager -> FB_VisionAlign -> Vision
				//
				// P1 = CameraID.
				// P2 = JobID.
				// P3 = A_Var index nhận business result.
				//
				// A_Var[P3] = 1 : Vision Result OK.
				// A_Var[P3] = 0 : Vision Result NG / NOT_FOUND / LOW_SCORE / ...
				//
				// Lỗi communication/config/protocol/timeout:
				// -> A_VisionError = TRUE.
				// -> Robot Blarm.
				// -> Không chuyển sang step tiếp theo.
				//=========================================================================
			
			
				//=========================================================================
				// 1. START COMMAND
				// Chỉ thực hiện một lần khi command Vision chưa active.
				//=========================================================================
				IF NOT xVisionStepActiveB THEN
			
					//---------------------------------------------------------------------
					// Latch tham số command.
					//---------------------------------------------------------------------
					uiVisionCameraIDB := INT_TO_UINT(step_PRG_B_Interpreter.P1);
					uiVisionJobIDB := INT_TO_UINT(step_PRG_B_Interpreter.P2);
					iVisionResultVarB := DINT_TO_INT(step_PRG_B_Interpreter.P3);
			
					//---------------------------------------------------------------------
					// Kiểm tra CameraID trước khi gửi Request.
					//---------------------------------------------------------------------
					IF (uiVisionCameraIDB < 1)
					OR (uiVisionCameraIDB > GVL.C_MAX_VISION_CHANNELS) THEN
			
						GVL.B_VisionDone := FALSE;
						GVL.B_VisionOK := FALSE;
						GVL.B_VisionError := TRUE;
			
						GVL.B_RunAlarm := TRUE;
						GVL.B_RunAlarmCode := 2201;
						GVL.B_RunErrorStep := GVL.B_RunStep;
						GVL.B_RunState := 900;
			
					//---------------------------------------------------------------------
					// A_Var của project hiện tại có index 0..200.
					//---------------------------------------------------------------------
					ELSIF (iVisionResultVarB < 0)
					OR (iVisionResultVarB > 200) THEN
			
						GVL.B_VisionDone := FALSE;
						GVL.B_VisionOK := FALSE;
						GVL.B_VisionError := TRUE;
			
						GVL.B_RunAlarm := TRUE;
						GVL.B_RunAlarmCode := 2202;
						GVL.B_RunErrorStep := GVL.B_RunStep;
						GVL.B_RunState := 900;
			
					ELSE
						//-----------------------------------------------------------------
						// Xóa business result cũ.
						//-----------------------------------------------------------------
						GVL.B_Var[iVisionResultVarB] := 0;
			
						//-----------------------------------------------------------------
						// Xóa status tương thích logic Robot cũ.
						//-----------------------------------------------------------------
						GVL.B_VisionDone := FALSE;
						GVL.B_VisionOK := FALSE;
						GVL.B_VisionError := FALSE;
			
						//-----------------------------------------------------------------
						// Gửi Request sang Vision Manager.
						//
						// CameraID và JobID phải được ghi TRƯỚC Execute.
						//-----------------------------------------------------------------
						GVL.g_stVisionAlignRequestB.CameraID := uiVisionCameraIDB;
						GVL.g_stVisionAlignRequestB.JobID := uiVisionJobIDB;
						GVL.g_stVisionAlignRequestB.Execute := TRUE;
			
						//-----------------------------------------------------------------
						// Đánh dấu command Vision của Robot B đang hoạt động.
						//-----------------------------------------------------------------
						xVisionStepActiveB := TRUE;
					END_IF;
				END_IF;
			
			
				//=========================================================================
				// 2. WAIT TRANSACTION DONE
				//=========================================================================
				IF xVisionStepActiveB AND GVL.g_stVisionAlignRequestB.Done THEN
			
					//---------------------------------------------------------------------
					// Vision transaction hoàn thành bình thường.
					//
					// ResultOK quyết định business result:
					// TRUE  -> A_Var[P3] = 1.
					// FALSE -> A_Var[P3] = 0.
					//---------------------------------------------------------------------
					IF GVL.g_stVisionAlignRequestB.ResultOK THEN
						GVL.B_Var[iVisionResultVarB] := 1;
						GVL.B_VisionOK := TRUE;
					ELSE
						GVL.B_Var[iVisionResultVarB] := 0;
						GVL.B_VisionOK := FALSE;
					END_IF;
			
					//---------------------------------------------------------------------
					// Transaction đã hoàn thành.
					//---------------------------------------------------------------------
					GVL.B_VisionDone := TRUE;
					GVL.B_VisionError := FALSE;
			
					//---------------------------------------------------------------------
					// Hạ Execute = ACK từ Robot về Manager.
					//
					// Manager thấy Execute FALSE sẽ:
					// - Reset Done.
					// - Giải phóng Camera.
					// - Đưa Camera về State 0.
					//---------------------------------------------------------------------
					GVL.g_stVisionAlignRequestB.Execute := FALSE;
			
					//---------------------------------------------------------------------
					// Kết thúc command local.
					//---------------------------------------------------------------------
					xVisionStepActiveB := FALSE;
			
					//---------------------------------------------------------------------
					// Chuyển sang command tiếp theo.
					//---------------------------------------------------------------------
					GVL.B_RunStep := GVL.B_RunStep + 1;
					GVL.B_RunState := 0;
			
					//---------------------------------------------------------------------
					// Step Mode: giữ chương trình sau khi hoàn thành một command.
					//---------------------------------------------------------------------
					IF GVL.B_RunMode = 1 THEN
						GVL.B_StepHold := TRUE;
					END_IF;
			
			
				//=========================================================================
				// 3. WAIT TRANSACTION ERROR
				//=========================================================================
				ELSIF xVisionStepActiveB AND GVL.g_stVisionAlignRequestB.Error THEN
				
					// LƯU MÃ LỖI TRƯỚC KHI HẠ EXECUTE.
					// Manager sẽ reset ErrorID sau khi Execute = FALSE.
					iVisionErrorIDB := GVL.g_stVisionAlignRequestB.ErrorID;
				
					// Không sử dụng kết quả Vision khi transaction lỗi.
					GVL.B_Var[iVisionResultVarB] := 0;
					GVL.B_VisionDone := FALSE;
					GVL.B_VisionOK := FALSE;
					GVL.B_VisionError := TRUE;
				
					// Báo Alarm Robot.
					GVL.B_RunAlarm := TRUE;
					GVL.B_RunAlarmCode := 2201;
					GVL.B_RunErrorStep := GVL.B_RunStep;
					GVL.B_RunState := 900;
				
					// Kết thúc command Vision local.
					xVisionStepActiveB := FALSE;
				
					// Hạ Execute CUỐI CÙNG.
					// Manager nhận ACK này và sau đó mới reset Request.
					GVL.g_stVisionAlignRequestB.Execute := FALSE;
				
				END_IF;
							
	
			E_RobotCmd.CMD_VISION_SET_POINT:

				//=========================================================================
				// VISION SET POINT
				//-------------------------------------------------------------------------
				// P1 = Master Point No.
				// P2 = Destination Point No.
				// P3 = Vision Result Index.
				//
				// Destination = Master + Vision Result[P3]
				//
				// Ví dụ:
				// VISION_SET_POINT P10 P101 1
				// VISION_SET_POINT P10 P102 2
				//
				// P101 = P10 + Result[1]
				// P102 = P10 + Result[2]
				//
				// Chỉ yêu cầu Header của Vision Result hợp lệ.
				// Không kiểm tra ObjectCount.
				// Không kiểm tra Object.Valid.
				// Không kiểm tra Vision có trả đủ số lượng Object hay không.
				//=========================================================================
			
				//-------------------------------------------------------------------------
				// 1. KIỂM TRA MASTER / DESTINATION POINT
				//-------------------------------------------------------------------------
				IF (step_PRG_B_Interpreter.P1 < 1) OR (step_PRG_B_Interpreter.P1 > 500)
				OR (step_PRG_B_Interpreter.P2 < 1) OR (step_PRG_B_Interpreter.P2 > 500)
				OR (step_PRG_B_Interpreter.P1 = step_PRG_B_Interpreter.P2) THEN
			
					GVL.B_RunAlarm := TRUE;
					GVL.B_RunAlarmCode := 2203;      // Master/Destination Point không hợp lệ.
					GVL.B_RunErrorStep := GVL.B_RunStep;
					GVL.B_RunState := 900;
			
				//-------------------------------------------------------------------------
				// 2. KIỂM TRA RESULT INDEX
				//-------------------------------------------------------------------------
				ELSIF (step_PRG_B_Interpreter.P3 < 1)
				OR (step_PRG_B_Interpreter.P3 > GVL.C_MAX_VISION_TRACK_OBJECTS_PER_FRAME) THEN
			
					GVL.B_RunAlarm := TRUE;
					GVL.B_RunAlarmCode := 2205;      // Vision Result Index ngoài vùng Array.
					GVL.B_RunErrorStep := GVL.B_RunStep;
					GVL.B_RunState := 900;
			
				//-------------------------------------------------------------------------
				// 3. CHỈ KIỂM TRA HEADER
				//-------------------------------------------------------------------------
				ELSIF NOT GVL.g_aVisionResult[uiVisionCameraIDB].Header.Valid THEN
			
					GVL.B_RunAlarm := TRUE;
					GVL.B_RunAlarmCode := 2204;      // Vision Header không hợp lệ.
					GVL.B_RunErrorStep := GVL.B_RunStep;
					GVL.B_RunState := 900;
			
				ELSE
			
					//=====================================================================
					// 4. DESTINATION = MASTER + VISION RESULT[P3]
					//=====================================================================
			
					// X
					GVL_1.DATA_RB_B.X_POS[DINT_TO_INT(step_PRG_B_Interpreter.P2)] :=
						GVL_1.DATA_RB_B.X_POS[DINT_TO_INT(step_PRG_B_Interpreter.P1)]
						+ GVL.g_aVisionResult[uiVisionCameraIDB].TrackObjectResult.Objects[DINT_TO_UINT(step_PRG_B_Interpreter.P3)].Pos.X;
			
					// Y
					GVL_1.DATA_RB_B.Y_POS[DINT_TO_INT(step_PRG_B_Interpreter.P2)] :=
						GVL_1.DATA_RB_B.Y_POS[DINT_TO_INT(step_PRG_B_Interpreter.P1)]
						+ GVL.g_aVisionResult[uiVisionCameraIDB].TrackObjectResult.Objects[DINT_TO_UINT(step_PRG_B_Interpreter.P3)].Pos.Y;
			
					// Z
					GVL_1.DATA_RB_B.Z_POS[DINT_TO_INT(step_PRG_B_Interpreter.P2)] :=
						GVL_1.DATA_RB_B.Z_POS[DINT_TO_INT(step_PRG_B_Interpreter.P1)]
						+ GVL.g_aVisionResult[uiVisionCameraIDB].TrackObjectResult.Objects[DINT_TO_UINT(step_PRG_B_Interpreter.P3)].Pos.Z;
			
					// R
					GVL_1.DATA_RB_B.R_POS[DINT_TO_INT(step_PRG_B_Interpreter.P2)] :=
						GVL_1.DATA_RB_B.R_POS[DINT_TO_INT(step_PRG_B_Interpreter.P1)]
						+ GVL.g_aVisionResult[uiVisionCameraIDB].TrackObjectResult.Objects[DINT_TO_UINT(step_PRG_B_Interpreter.P3)].Pos.A;
			
					//=====================================================================
					// 5. COMMAND HOÀN THÀNH
					//=====================================================================
					GVL.B_RunStep := GVL.B_RunStep + 1;
					GVL.B_RunState := 0;
			
					IF GVL.B_RunMode = 1 THEN
						GVL.B_StepHold := TRUE;
					END_IF;
			
				END_IF;
	
	
			E_RobotCmd.CMD_VISION_PICK:

				//=========================================================================
				// VISION PICK
				//-------------------------------------------------------------------------
				// Hiện tại mới xác nhận Result Vision tồn tại.
				// Phần Camera->Robot Transform và tạo Target Pick sẽ bổ sung sau.
				//=========================================================================
			
				IF GVL.B_VisionHeaderOK THEN
					GVL.B_RunStep := GVL.B_RunStep + 1;
					GVL.B_RunState := 0;
			
					IF GVL.B_RunMode = 1 THEN
						GVL.B_StepHold := TRUE;
					END_IF;
			
				ELSE
					GVL.B_RunAlarm := TRUE;
					GVL.B_RunAlarmCode := 2202;
					GVL.B_RunErrorStep := GVL.B_RunStep;
					GVL.B_RunState := 900;
				END_IF;
	
	
			E_RobotCmd.CMD_VISION_CHECK:

				//=========================================================================
				// CHECK LAST VISION RESULT
				//-------------------------------------------------------------------------
				// TRUE  -> chạy Step tiếp theo.
				// FALSE -> nhảy tới ELSE / END_IF.
				//=========================================================================
			
				IF GVL.B_VisionHeaderOK THEN
					GVL.B_RunStep := GVL.B_RunStep + 1;
				ELSE
					GVL.B_RunStep := F_FindElseOrEndIf_B(GVL.B_RunStep);
				END_IF;
			
				GVL.B_RunState := 0;
			
				IF GVL.B_RunMode = 1 THEN
					GVL.B_StepHold := TRUE;
				END_IF;
			
			//================================================
			// TRACKING
			//================================================
			E_RobotCmd.CMD_TRACK_ON:
				GVL.B_TrackEnable := TRUE;
				GVL.B_RunStep := GVL.B_RunStep + 1;
				GVL.B_RunState := 0;
	
	
			E_RobotCmd.CMD_TRACK_OFF:
				GVL.B_TrackEnable := FALSE;
				GVL.B_RunStep := GVL.B_RunStep + 1;
				GVL.B_RunState := 0;
	
	
			//==========================================================================
			// TRACK PICK
			//--------------------------------------------------------------------------
			// P1 = RecipeID
			// P2 = Target Pick Count
			// P3 = Tool Mask
			//
			// Ví dụ:
			// P1=1, P2=1, P3=1 -> Recipe 1, Pick 1, chỉ Tool 1.
			// P1=1, P2=2, P3=3 -> Recipe 1, Pick 2, Tool 1 + Tool 2.
			//==========================================================================
			E_RobotCmd.CMD_TRACK_PICK:
			
				//----------------------------------------------------------------------
				// 1. CHỈ PHÁT COMMAND MỘT LẦN
				//----------------------------------------------------------------------
				IF NOT GVL.B_StepActive THEN
			
					// Chỉ bắt đầu khi Motion Pipeline trước đó đã sạch.
					IF (GVL.B_MotionCount <= 0)
					AND (GVL.B_ActiveMotionCount <= 0)
					AND NOT GVL.B_MotionManagerBusy THEN
			
						//--------------------------------------------------------------
						// Tạo CommandID mới.
						//--------------------------------------------------------------
						GVL.g_stMultiTrackCommandB.CommandID :=
							GVL.g_stMultiTrackCommandB.CommandID + 1;
			
						IF GVL.g_stMultiTrackCommandB.CommandID = 0 THEN
							GVL.g_stMultiTrackCommandB.CommandID := 1;
						END_IF;
			
						//--------------------------------------------------------------
						// Nạp tham số từ dòng Interpreter.
						//--------------------------------------------------------------
						GVL.g_stMultiTrackCommandB.RecipeID :=
							INT_TO_UINT(step_PRG_B_Interpreter.P1);
			
						GVL.g_stMultiTrackCommandB.TargetPickCountOverride :=
							INT_TO_UINT(step_PRG_B_Interpreter.P2);
			
						GVL.g_stMultiTrackCommandB.ToolMaskOverride :=
							DINT_TO_DWORD(step_PRG_B_Interpreter.P3);
			
						//--------------------------------------------------------------
						// Command mới.
						//--------------------------------------------------------------
						GVL.g_stMultiTrackCommandB.Reset := FALSE;
						GVL.g_stMultiTrackCommandB.Abort := FALSE;
						GVL.g_stMultiTrackCommandB.Execute := TRUE;
			
						//--------------------------------------------------------------
						// Nhớ CommandID mà Interpreter đang chờ.
						//--------------------------------------------------------------
						udiTrackCommandIDB :=
							GVL.g_stMultiTrackCommandB.CommandID;
			
						//--------------------------------------------------------------
						// Không phát lại command ở scan tiếp theo.
						//--------------------------------------------------------------
						GVL.B_StepActive := TRUE;
			
					END_IF;
			
				END_IF;
			
			
				//----------------------------------------------------------------------
				// 2. TRACKING HOÀN THÀNH ĐÚNG COMMAND
				//----------------------------------------------------------------------
				IF GVL.B_StepActive
				AND GVL.g_xTrackOKB
				AND GVL.g_udiTrackDoneCommandIDB = udiTrackCommandIDB THEN
			
					// Hạ Execute sau khi Application hoàn thành.
					GVL.g_stMultiTrackCommandB.Execute := FALSE;
			
					// Kết thúc transaction của Interpreter.
					GVL.B_StepActive := FALSE;
					udiTrackCommandIDB := 0;
			
					// Sang dòng chương trình tiếp theo.
					GVL.B_RunStep := GVL.B_RunStep + 1;
					GVL.B_RunState := 0;
			
					// Step Mode: dừng sau khi hoàn thành TRACK_PICK.
					IF GVL.B_RunMode = 1 THEN
						GVL.B_StepHold := TRUE;
					END_IF;
			
				//----------------------------------------------------------------------
				// 3. TRACKING ERROR
				//----------------------------------------------------------------------
				ELSIF GVL.B_StepActive
				AND GVL.g_xTrackErrorB THEN
			
					GVL.g_stMultiTrackCommandB.Execute := FALSE;
			
					GVL.B_StepActive := FALSE;
					udiTrackCommandIDB := 0;
			
					GVL.B_RunAlarm := TRUE;
					GVL.B_RunAlarmCode :=
						UDINT_TO_INT(GVL.g_udiTrackErrorIDB);
			
					GVL.B_RunErrorStep := GVL.B_RunStep;
					GVL.B_RunState := 900;
			
				END_IF;
			
			//=========================================================================
			// TOOL RELEASE
			//-------------------------------------------------------------------------
			// P1 = ToolID cần nhả sản phẩm.
			//=========================================================================
			E_RobotCmd.CMD_TOOL_RELEASE:
			
				//---------------------------------------------------------------------
				// 1. PHÁT LỆNH RELEASE MỘT LẦN
				//---------------------------------------------------------------------
				IF NOT GVL.B_StepActive THEN
			
					// Kiểm tra ToolID hợp lệ.
					IF (step_PRG_B_Interpreter.P1 >= 1)
					AND (step_PRG_B_Interpreter.P1 <= GVL.C_MAX_TOOLS) THEN
			
						//-------------------------------------------------------------
						// Chỉ Release Tool đang thực sự giữ sản phẩm.
						//-------------------------------------------------------------
						IF GVL.g_aToolStatusB[step_PRG_B_Interpreter.P1].Occupied THEN
			
							//---------------------------------------------------------
							// Tạo CommandID mới.
							//---------------------------------------------------------
							GVL.g_stInterpreterToolCommandB.CommandID :=
								GVL.g_stInterpreterToolCommandB.CommandID + 1;
			
							IF GVL.g_stInterpreterToolCommandB.CommandID = 0 THEN
								GVL.g_stInterpreterToolCommandB.CommandID := 1;
							END_IF;
			
							//---------------------------------------------------------
							// Nạp command.
							//---------------------------------------------------------
							GVL.g_stInterpreterToolCommandB.ToolID :=
								INT_TO_UINT(step_PRG_B_Interpreter.P1);
			
							GVL.g_stInterpreterToolCommandB.CommandType :=
								E_ToolCommandType.RELEASE;
			
							// Giữ ObjectID hiện tại để debug/trace.
							GVL.g_stInterpreterToolCommandB.ObjectID :=
								GVL.g_aToolStatusB[step_PRG_B_Interpreter.P1].HeldObjectID;
			
							GVL.g_stInterpreterToolCommandB.Reset := FALSE;
							GVL.g_stInterpreterToolCommandB.Abort := FALSE;
							GVL.g_stInterpreterToolCommandB.Execute := TRUE;
			
							//---------------------------------------------------------
							// Nhớ CommandID đang chờ.
							//---------------------------------------------------------
							udiToolReleaseCommandIDB :=
								GVL.g_stInterpreterToolCommandB.CommandID;
			
							GVL.B_StepActive := TRUE;
			
						ELSE
			
							//---------------------------------------------------------
							// Tool không giữ vật -> coi là lỗi dạy chương trình.
							//---------------------------------------------------------
							GVL.B_RunAlarm := TRUE;
							GVL.B_RunAlarmCode := 2502;
							GVL.B_RunErrorStep := GVL.B_RunStep;
							GVL.B_RunState := 900;
			
						END_IF;
			
					ELSE
			
						//-------------------------------------------------------------
						// ToolID ngoài phạm vi.
						//-------------------------------------------------------------
						GVL.B_RunAlarm := TRUE;
						GVL.B_RunAlarmCode := 2501;
						GVL.B_RunErrorStep := GVL.B_RunStep;
						GVL.B_RunState := 900;
			
					END_IF;
			
				END_IF;
			
			
				//---------------------------------------------------------------------
				// 2. RELEASE HOÀN THÀNH
				//---------------------------------------------------------------------
				IF GVL.B_StepActive
				AND GVL.g_aToolStatusB[step_PRG_B_Interpreter.P1].Done
				AND GVL.g_aToolStatusB[step_PRG_B_Interpreter.P1].ResponseCommandID
					= udiToolReleaseCommandIDB THEN
			
					//-------------------------------------------------------------
					// Hạ Execute để tạo lại cạnh cho command sau.
					//-------------------------------------------------------------
					GVL.g_stInterpreterToolCommandB.Execute := FALSE;
			
					GVL.B_StepActive := FALSE;
					udiToolReleaseCommandIDB := 0;
			
					//-------------------------------------------------------------
					// Sang step kế tiếp.
					//-------------------------------------------------------------
					GVL.B_RunStep := GVL.B_RunStep + 1;
					GVL.B_RunState := 0;
			
					IF GVL.B_RunMode = 1 THEN
						GVL.B_StepHold := TRUE;
					END_IF;
			
			
				//---------------------------------------------------------------------
				// 3. TOOL ERROR
				//---------------------------------------------------------------------
				ELSIF GVL.B_StepActive
				AND GVL.g_aToolStatusB[step_PRG_B_Interpreter.P1].Error THEN
			
					GVL.g_stInterpreterToolCommandB.Execute := FALSE;
			
					GVL.B_StepActive := FALSE;
					udiToolReleaseCommandIDB := 0;
			
					GVL.B_RunAlarm := TRUE;
			
					GVL.B_RunAlarmCode :=
						UDINT_TO_INT(
							GVL.g_aToolStatusB[step_PRG_B_Interpreter.P1].ErrorID
						);
			
					GVL.B_RunErrorStep := GVL.B_RunStep;
					GVL.B_RunState := 900;
			
				END_IF;
	

			E_RobotCmd.CMD_TRACK_PLACE:
				GVL.B_TrackPlaceReq := TRUE;
	
				IF GVL.B_TrackPlaceDone THEN
					GVL.B_TrackPlaceReq := FALSE;
					GVL.B_RunStep := GVL.B_RunStep + 1;
					GVL.B_RunState := 0;
				END_IF;
				
			E_RobotCmd.CMD_CONV_PICK:

// 				// Không bắt đầu Application khi pipeline motion cũ còn hoạt động.
// 				IF NOT GVL.B_StepActive THEN
// 					IF GVL.B_MotionCount = 0 AND GVL.B_ActiveMotionCount = 0 THEN
// 						GVL.g_stApplicationCommandB.ApplicationID := E_ApplicationID.APP_CONVEYOR_PICK;
// 						GVL.g_stApplicationCommandB.RecipeID := TO_UINT(step.P1);
// 						GVL.g_stApplicationCommandB.RobotID := 1;
// 						GVL.g_stApplicationCommandB.CommandID := GVL.g_stApplicationCommandB.CommandID + 1;
// 						GVL.g_stApplicationCommandB.Execute := TRUE;
// 						GVL.B_StepActive := TRUE;
// 					END_IF;
// 				END_IF;
// 			
// 				// Application hoàn thành: hạ Execute và chuyển step.
// 				IF GVL.g_stApplicationResponseB.Done THEN
// 					GVL.g_stApplicationCommandB.Execute := FALSE;
// 					GVL.B_StepActive := FALSE;
// 					GVL.B_RunStep := GVL.B_RunStep + 1;
// 				END_IF;
// 			
// 				// Application lỗi: dừng Interpreter.
// 				IF GVL.g_stApplicationResponseB.Error THEN
// 					GVL.g_stApplicationCommandB.Execute := FALSE;
// 					GVL.B_StepActive := FALSE;
// 					GVL.B_RunAlarm := TRUE;
// 					GVL.B_RunAlarmCode := TO_INT(GVL.g_stApplicationResponseB.ErrorID);
// 					GVL.B_RunErrorStep := GVL.B_RunStep;
// 				END_IF;

				// Chỉ bắt đầu khi Motion Queue và các slot hiện tại đã sạch.
				IF NOT GVL.B_StepActive THEN
					IF GVL.B_MotionCount = 0 AND GVL.B_ActiveMotionCount = 0 THEN
						GVL.B_TrackStartCmd := TRUE;
						GVL.B_StepActive := TRUE;
					END_IF;
				END_IF;
			
				// Sau khi engine nhận cạnh Start, hạ request.
				IF GVL.B_TrackEngineBusy THEN
					GVL.B_TrackStartCmd := FALSE;
				END_IF;
			
				// Hoàn thành application thì tăng step.
				IF GVL.B_TrackEngineDone THEN
					GVL.B_TrackStartCmd := FALSE;
					GVL.B_StepActive := FALSE;
					GVL.B_RunStep := GVL.B_RunStep + 1;
					GVL.B_RunState := 0;
				END_IF;
			
				// Lỗi application thì dừng Interpreter.
				IF GVL.B_TrackEngineError THEN
					GVL.B_TrackStartCmd := FALSE;
					GVL.B_StepActive := FALSE;
					GVL.B_RunAlarm := TRUE;
					GVL.B_RunAlarmCode := TO_INT(GVL.B_TrackEngineErrorID);
					GVL.B_RunErrorStep := GVL.B_RunStep;
				END_IF;

			//=========================================================================
			// MODBUS / POINT COMMANDS - ROBOT B
			//=========================================================================
			
			E_RobotCmd.CMD_MB_REG_READ:
				// P1 = MODBUS Index [0..1999]
				// P2 = B_Reg Destination [1..200]
				// GVL.MODBUS[] dùng chung
				// Giá trị MODBUS được hiểu là INT16 có dấu
			
				IF (step_PRG_B_Interpreter.P1 >= 0) AND (step_PRG_B_Interpreter.P1 <= 1999)
				AND (step_PRG_B_Interpreter.P2 >= 1) AND (step_PRG_B_Interpreter.P2 <= 200) THEN
			
					GVL.B_Reg[step_PRG_B_Interpreter.P2] := INT_TO_DINT(WORD_TO_INT(GVL.MODBUS[step_PRG_B_Interpreter.P1]));
			
					GVL.B_RunStep := GVL.B_RunStep + 1;
					GVL.B_RunState := 0;
					IF GVL.B_RunMode = 1 THEN GVL.B_StepHold := TRUE; END_IF;
			
				ELSE
					GVL.B_RunAlarm := TRUE;
					GVL.B_RunAlarmCode := 2503;
					GVL.B_RunErrorStep := GVL.B_RunStep;
					GVL.B_RunState := 900;
				END_IF;
	
			
			E_RobotCmd.CMD_MB_REG_SET:
				// P1 = MODBUS Index [0..1999]
				// P2 = Signed INT16 value
				IF (step_PRG_B_Interpreter.P1 >= 0) AND (step_PRG_B_Interpreter.P1 <= 1999) THEN
					GVL.MODBUS[step_PRG_B_Interpreter.P1] := INT_TO_WORD(step_PRG_B_Interpreter.P2);
			
					GVL.B_RunStep := GVL.B_RunStep + 1;
					GVL.B_RunState := 0;
					IF GVL.B_RunMode = 1 THEN GVL.B_StepHold := TRUE; END_IF;
				ELSE
					GVL.B_RunAlarm := TRUE;
					GVL.B_RunAlarmCode := 2501;
					GVL.B_RunErrorStep := GVL.B_RunStep;
					GVL.B_RunState := 900;
				END_IF;
			
			
			E_RobotCmd.CMD_MB_BIT_SET:
				// P1 = MODBUS Index [0..1999]
				// P2 = Bit Index [0..15]
				// P3 = 0: Reset / <>0: Set
				IF (step_PRG_B_Interpreter.P1 >= 0) AND (step_PRG_B_Interpreter.P1 <= 1999)
				AND (step_PRG_B_Interpreter.P2 >= 0) AND (step_PRG_B_Interpreter.P2 <= 15) THEN
			
					IF step_PRG_B_Interpreter.P3 <> 0 THEN
						GVL.MODBUS[step_PRG_B_Interpreter.P1] := GVL.MODBUS[step_PRG_B_Interpreter.P1] OR SHL(WORD#1, step_PRG_B_Interpreter.P2);
					ELSE
						GVL.MODBUS[step_PRG_B_Interpreter.P1] := GVL.MODBUS[step_PRG_B_Interpreter.P1] AND NOT SHL(WORD#1, step_PRG_B_Interpreter.P2);
					END_IF;
			
					GVL.B_RunStep := GVL.B_RunStep + 1;
					GVL.B_RunState := 0;
					IF GVL.B_RunMode = 1 THEN GVL.B_StepHold := TRUE; END_IF;
				ELSE
					GVL.B_RunAlarm := TRUE;
					GVL.B_RunAlarmCode := 2502;
					GVL.B_RunErrorStep := GVL.B_RunStep;
					GVL.B_RunState := 900;
				END_IF;
			
			//=========================================================================
			// POINT CALCULATION COMMANDS - ROBOT B
			//=========================================================================
			
			E_RobotCmd.CMD_POINT_COPY:
				// P1 = Destination Point
				// P2 = Source Point
				IF (step_PRG_B_Interpreter.P1 >= 1) AND (step_PRG_B_Interpreter.P1 <= 500)
				AND (step_PRG_B_Interpreter.P2 >= 1) AND (step_PRG_B_Interpreter.P2 <= 500) THEN
					GVL_1.DATA_RB_B.X_POS[step_PRG_B_Interpreter.P1] := GVL_1.DATA_RB_B.X_POS[step_PRG_B_Interpreter.P2];
					GVL_1.DATA_RB_B.Y_POS[step_PRG_B_Interpreter.P1] := GVL_1.DATA_RB_B.Y_POS[step_PRG_B_Interpreter.P2];
					GVL_1.DATA_RB_B.Z_POS[step_PRG_B_Interpreter.P1] := GVL_1.DATA_RB_B.Z_POS[step_PRG_B_Interpreter.P2];
					GVL_1.DATA_RB_B.R_POS[step_PRG_B_Interpreter.P1] := GVL_1.DATA_RB_B.R_POS[step_PRG_B_Interpreter.P2];
					GVL.B_RunStep := GVL.B_RunStep + 1;
					GVL.B_RunState := 0;
					IF GVL.B_RunMode = 1 THEN GVL.B_StepHold := TRUE; END_IF;
				ELSE
					GVL.B_RunAlarm := TRUE;
					GVL.B_RunAlarmCode := 2510;
					GVL.B_RunErrorStep := GVL.B_RunStep;
					GVL.B_RunState := 900;
				END_IF;
			
			
			E_RobotCmd.CMD_POINT_ADD:
				// P1 = Destination Point
				// P2 = Base Point
				// P3 = Offset Point
				IF (step_PRG_B_Interpreter.P1 >= 1) AND (step_PRG_B_Interpreter.P1 <= 500)
				AND (step_PRG_B_Interpreter.P2 >= 1) AND (step_PRG_B_Interpreter.P2 <= 500)
				AND (step_PRG_B_Interpreter.P3 >= 1) AND (step_PRG_B_Interpreter.P3 <= 500) THEN
					GVL_1.DATA_RB_B.X_POS[step_PRG_B_Interpreter.P1] := GVL_1.DATA_RB_B.X_POS[step_PRG_B_Interpreter.P2] + GVL_1.DATA_RB_B.X_POS[step_PRG_B_Interpreter.P3];
					GVL_1.DATA_RB_B.Y_POS[step_PRG_B_Interpreter.P1] := GVL_1.DATA_RB_B.Y_POS[step_PRG_B_Interpreter.P2] + GVL_1.DATA_RB_B.Y_POS[step_PRG_B_Interpreter.P3];
					GVL_1.DATA_RB_B.Z_POS[step_PRG_B_Interpreter.P1] := GVL_1.DATA_RB_B.Z_POS[step_PRG_B_Interpreter.P2] + GVL_1.DATA_RB_B.Z_POS[step_PRG_B_Interpreter.P3];
					GVL_1.DATA_RB_B.R_POS[step_PRG_B_Interpreter.P1] := GVL_1.DATA_RB_B.R_POS[step_PRG_B_Interpreter.P2] + GVL_1.DATA_RB_B.R_POS[step_PRG_B_Interpreter.P3];
					GVL.B_RunStep := GVL.B_RunStep + 1;
					GVL.B_RunState := 0;
					IF GVL.B_RunMode = 1 THEN GVL.B_StepHold := TRUE; END_IF;
				ELSE
					GVL.B_RunAlarm := TRUE;
					GVL.B_RunAlarmCode := 2511;
					GVL.B_RunErrorStep := GVL.B_RunStep;
					GVL.B_RunState := 900;
				END_IF;
			
			
			E_RobotCmd.CMD_POINT_SUB:
				// P1 = Destination Point
				// P2 = Base Point
				// P3 = Offset Point
				IF (step_PRG_B_Interpreter.P1 >= 1) AND (step_PRG_B_Interpreter.P1 <= 500)
				AND (step_PRG_B_Interpreter.P2 >= 1) AND (step_PRG_B_Interpreter.P2 <= 500)
				AND (step_PRG_B_Interpreter.P3 >= 1) AND (step_PRG_B_Interpreter.P3 <= 500) THEN
					GVL_1.DATA_RB_B.X_POS[step_PRG_B_Interpreter.P1] := GVL_1.DATA_RB_B.X_POS[step_PRG_B_Interpreter.P2] - GVL_1.DATA_RB_B.X_POS[step_PRG_B_Interpreter.P3];
					GVL_1.DATA_RB_B.Y_POS[step_PRG_B_Interpreter.P1] := GVL_1.DATA_RB_B.Y_POS[step_PRG_B_Interpreter.P2] - GVL_1.DATA_RB_B.Y_POS[step_PRG_B_Interpreter.P3];
					GVL_1.DATA_RB_B.Z_POS[step_PRG_B_Interpreter.P1] := GVL_1.DATA_RB_B.Z_POS[step_PRG_B_Interpreter.P2] - GVL_1.DATA_RB_B.Z_POS[step_PRG_B_Interpreter.P3];
					GVL_1.DATA_RB_B.R_POS[step_PRG_B_Interpreter.P1] := GVL_1.DATA_RB_B.R_POS[step_PRG_B_Interpreter.P2] - GVL_1.DATA_RB_B.R_POS[step_PRG_B_Interpreter.P3];
					GVL.B_RunStep := GVL.B_RunStep + 1;
					GVL.B_RunState := 0;
					IF GVL.B_RunMode = 1 THEN GVL.B_StepHold := TRUE; END_IF;
				ELSE
					GVL.B_RunAlarm := TRUE;
					GVL.B_RunAlarmCode := 2512;
					GVL.B_RunErrorStep := GVL.B_RunStep;
					GVL.B_RunState := 900;
				END_IF;
			
			
			E_RobotCmd.CMD_POINT_ADD_VALUE:
				// P1 = Point cần thay đổi
				// P2=X, P3=Y, P4=Z, P5=R
				IF (step_PRG_B_Interpreter.P1 >= 1) AND (step_PRG_B_Interpreter.P1 <= 500) THEN
					GVL_1.DATA_RB_B.X_POS[step_PRG_B_Interpreter.P1] := GVL_1.DATA_RB_B.X_POS[step_PRG_B_Interpreter.P1] + INT_TO_REAL(step_PRG_B_Interpreter.P2)/1000;
					GVL_1.DATA_RB_B.Y_POS[step_PRG_B_Interpreter.P1] := GVL_1.DATA_RB_B.Y_POS[step_PRG_B_Interpreter.P1] + DINT_TO_REAL(step_PRG_B_Interpreter.P3)/1000;
					GVL_1.DATA_RB_B.Z_POS[step_PRG_B_Interpreter.P1] := GVL_1.DATA_RB_B.Z_POS[step_PRG_B_Interpreter.P1] + INT_TO_REAL(step_PRG_B_Interpreter.P4)/1000;
					GVL_1.DATA_RB_B.R_POS[step_PRG_B_Interpreter.P1] := GVL_1.DATA_RB_B.R_POS[step_PRG_B_Interpreter.P1] + INT_TO_REAL(step_PRG_B_Interpreter.P5)/1000;
					GVL.B_RunStep := GVL.B_RunStep + 1;
					GVL.B_RunState := 0;
					IF GVL.B_RunMode = 1 THEN GVL.B_StepHold := TRUE; END_IF;
				ELSE
					GVL.B_RunAlarm := TRUE;
					GVL.B_RunAlarmCode := 2513;
					GVL.B_RunErrorStep := GVL.B_RunStep;
					GVL.B_RunState := 900;
				END_IF;
			
			
			E_RobotCmd.CMD_POINT_ADD_REG:
				// P1 = Point cần thay đổi
				// P2=RegX, P3=RegY, P4=RegZ, P5=RegR
				IF (step_PRG_B_Interpreter.P1 >= 1) AND (step_PRG_B_Interpreter.P1 <= 500)
				AND (step_PRG_B_Interpreter.P2 >= 1) AND (step_PRG_B_Interpreter.P2 <= 200)
				AND (step_PRG_B_Interpreter.P3 >= 1) AND (step_PRG_B_Interpreter.P3 <= 200)
				AND (step_PRG_B_Interpreter.P4 >= 1) AND (step_PRG_B_Interpreter.P4 <= 200)
				AND (step_PRG_B_Interpreter.P5 >= 1) AND (step_PRG_B_Interpreter.P5 <= 200) THEN
					GVL_1.DATA_RB_B.X_POS[step_PRG_B_Interpreter.P1] := GVL_1.DATA_RB_B.X_POS[step_PRG_B_Interpreter.P1] + DINT_TO_REAL(GVL.B_Reg[step_PRG_B_Interpreter.P2])/1000;
					GVL_1.DATA_RB_B.Y_POS[step_PRG_B_Interpreter.P1] := GVL_1.DATA_RB_B.Y_POS[step_PRG_B_Interpreter.P1] + DINT_TO_REAL(GVL.B_Reg[step_PRG_B_Interpreter.P3])/1000;
					GVL_1.DATA_RB_B.Z_POS[step_PRG_B_Interpreter.P1] := GVL_1.DATA_RB_B.Z_POS[step_PRG_B_Interpreter.P1] + DINT_TO_REAL(GVL.B_Reg[step_PRG_B_Interpreter.P4])/1000;
					GVL_1.DATA_RB_B.R_POS[step_PRG_B_Interpreter.P1] := GVL_1.DATA_RB_B.R_POS[step_PRG_B_Interpreter.P1] + DINT_TO_REAL(GVL.B_Reg[step_PRG_B_Interpreter.P5])/1000;
					GVL.B_RunStep := GVL.B_RunStep + 1;
					GVL.B_RunState := 0;
					IF GVL.B_RunMode = 1 THEN GVL.B_StepHold := TRUE; END_IF;
				ELSE
					GVL.B_RunAlarm := TRUE;
					GVL.B_RunAlarmCode := 2514;
					GVL.B_RunErrorStep := GVL.B_RunStep;
					GVL.B_RunState := 900;
				END_IF;
			
			
			E_RobotCmd.CMD_POINT_ADD_MB_REG:
				// P1 = Point cần thay đổi
				// P2=MB_X, P3=MB_Y, P4=MB_Z, P5=MB_R
				// MODBUS value = INT16 signed
				IF (step_PRG_B_Interpreter.P1 >= 1) AND (step_PRG_B_Interpreter.P1 <= 500)
				AND (step_PRG_B_Interpreter.P2 >= 0) AND (step_PRG_B_Interpreter.P2 <= 1999)
				AND (step_PRG_B_Interpreter.P3 >= 0) AND (step_PRG_B_Interpreter.P3 <= 1999)
				AND (step_PRG_B_Interpreter.P4 >= 0) AND (step_PRG_B_Interpreter.P4 <= 1999)
				AND (step_PRG_B_Interpreter.P5 >= 0) AND (step_PRG_B_Interpreter.P5 <= 1999) THEN
					GVL_1.DATA_RB_B.X_POS[step_PRG_B_Interpreter.P1] := GVL_1.DATA_RB_B.X_POS[step_PRG_B_Interpreter.P1] + INT_TO_REAL(WORD_TO_INT(GVL.MODBUS[step_PRG_B_Interpreter.P2]))/1000;
					GVL_1.DATA_RB_B.Y_POS[step_PRG_B_Interpreter.P1] := GVL_1.DATA_RB_B.Y_POS[step_PRG_B_Interpreter.P1] + INT_TO_REAL(WORD_TO_INT(GVL.MODBUS[step_PRG_B_Interpreter.P3]))/1000;
					GVL_1.DATA_RB_B.Z_POS[step_PRG_B_Interpreter.P1] := GVL_1.DATA_RB_B.Z_POS[step_PRG_B_Interpreter.P1] + INT_TO_REAL(WORD_TO_INT(GVL.MODBUS[step_PRG_B_Interpreter.P4]))/1000;
					GVL_1.DATA_RB_B.R_POS[step_PRG_B_Interpreter.P1] := GVL_1.DATA_RB_B.R_POS[step_PRG_B_Interpreter.P1] + INT_TO_REAL(WORD_TO_INT(GVL.MODBUS[step_PRG_B_Interpreter.P5]))/1000;
					GVL.B_RunStep := GVL.B_RunStep + 1;
					GVL.B_RunState := 0;
					IF GVL.B_RunMode = 1 THEN GVL.B_StepHold := TRUE; END_IF;
				ELSE
					GVL.B_RunAlarm := TRUE;
					GVL.B_RunAlarmCode := 2515;
					GVL.B_RunErrorStep := GVL.B_RunStep;
					GVL.B_RunState := 900;
				END_IF;
			
	
				
			E_RobotCmd.CMD_REG_SET,
			E_RobotCmd.CMD_REG_ADD,
			E_RobotCmd.CMD_REG_SUB,
			E_RobotCmd.CMD_REG_MUL,
			E_RobotCmd.CMD_REG_DIV,
			E_RobotCmd.CMD_REG_MOD:
			
				// P1 = Reg đích
				// P2 = SourceMode
				// P3 = Value hoặc Reg A
				// P4 = Reg B
			
				IF (step_PRG_B_Interpreter.P1 >= 1) AND (step_PRG_B_Interpreter.P1 <= 200) THEN
			
					GVL.B_Reg[step_PRG_B_Interpreter.P1] :=
						F_CalcReg_B(
							Cmd        := step_PRG_B_Interpreter.Cmd,
							DestReg    := step_PRG_B_Interpreter.P1,
							SourceMode := step_PRG_B_Interpreter.P2,
							P3         := step_PRG_B_Interpreter.P3,
							P4         := step_PRG_B_Interpreter.P4
						);
			
					GVL.B_RunStep := GVL.B_RunStep + 1;
					GVL.B_RunState := 0;
					// Nếu đang Step Mode thì dừng chờ sau khi chạy xong 1 lệnh
					IF GVL.B_RunMode = 1 THEN
						GVL.B_StepHold := TRUE;
					END_IF;
			
				ELSE
					GVL.B_RunAlarm := TRUE;
					GVL.B_RunAlarmCode := 2401; // Reg index invalid
					GVL.B_RunErrorStep := GVL.B_RunStep;
					GVL.B_RunState := 900;
				END_IF;
				
				
			E_RobotCmd.CMD_VAR_SET,
			E_RobotCmd.CMD_VAR_ADD,
			E_RobotCmd.CMD_VAR_SUB,
			E_RobotCmd.CMD_VAR_MUL,
			E_RobotCmd.CMD_VAR_DIV,
			E_RobotCmd.CMD_VAR_MOD:
				// P1 = Var đích
				// P2 = SourceMode
				// P3 = Value hoặc Var A
				// P4 = Var B
				IF (step_PRG_B_Interpreter.P1 >= 1) AND (step_PRG_B_Interpreter.P1 <= 200) THEN
			
					GVL.B_Var[step_PRG_B_Interpreter.P1] :=
						F_CalcVar_B(
							Cmd        := step_PRG_B_Interpreter.Cmd,
							DestVar    := step_PRG_B_Interpreter.P1,
							SourceMode := step_PRG_B_Interpreter.P2,
							P3         := step_PRG_B_Interpreter.P3,
							P4         := step_PRG_B_Interpreter.P4
						);
			
					GVL.B_RunStep := GVL.B_RunStep + 1;
					GVL.B_RunState := 0;
					// Nếu đang Step Mode thì dừng chờ sau khi chạy xong 1 lệnh
					IF GVL.B_RunMode = 1 THEN
						GVL.B_StepHold := TRUE;
					END_IF;
			
				ELSE
					GVL.B_RunAlarm := TRUE;
					GVL.B_RunAlarmCode := 2402;
					GVL.B_RunErrorStep := GVL.B_RunStep;
					GVL.B_RunState := 900;
				END_IF;
				
				
            E_RobotCmd.CMD_END:
                GVL.B_RunBusy := FALSE;
                GVL.B_RunDone := TRUE;
                GVL.B_RunState := 0;
		

        ELSE
            // Lệnh chưa hỗ trợ
            GVL.B_RunAlarm := TRUE;
            GVL.B_RunAlarmCode := 2001;
            GVL.B_RunErrorStep := GVL.B_RunStep;
            GVL.B_RunState := 900;
        END_CASE;


    100: // FILL PIPELINE

        // Nạp trước motion nếu:
        // 1. Chưa hết chương trình
        // 2. Step tiếp theo vẫn là motion
        // 3. Tổng số motion đang chờ + đang chạy chưa vượt pipeline depth
        IF (GVL.B_PipelineNextPushStep <= GVL.B_LengthStep)
           AND F_IsMotionCmd(GVL_1.Step_Cr_B[GVL.B_PipelineNextPushStep].Cmd)
           AND ((GVL.B_MotionCount + GVL.B_ActiveMotionCount) < GVL.B_PipelineDepth)
		   // AND (GVL.B_PipelineUsedCount < GVL.B_PipelineDepth)
        THEN
            GVL.B_PushMotionItem := F_BuildMotionItem_B(GVL.B_PipelineNextPushStep);
            GVL.B_PushMotionReq := TRUE;

            GVL.B_RunState := 110;
        ELSE
            // Pipeline đã đầy hoặc gặp lệnh logic
            GVL.B_RunState := 120;
        END_IF;


    110: // WAIT PUSH DONE
		
			IF GVL.B_PushMotionDone THEN
			
					GVL.B_PushMotionReq := FALSE;
					GVL.B_PushMotionDone := FALSE;
					
					//------------------------------------------------
					// Một motion chính thức thuộc pipeline
					//------------------------------------------------
					GVL.B_PipelineUsedCount :=
						GVL.B_PipelineUsedCount + 1;
			
					GVL.B_PipelineNextPushStep :=
						GVL.B_PipelineNextPushStep + 1;

					// Chờ motion hiện tại hoàn thành
					//GVL.B_RunState := 120;
					//GVL.B_RunState := 100;
					//------------------------------------------------
					// Kiểm tra BlendMode của Motion hiện tại
					//
					// P3:
					// 0  = Không Blending
					// >0 = Có Blending
					//------------------------------------------------
					
					IF GVL.B_RunMode = 0 THEN
						//IF (GVL_1.Step_Cr_B[GVL.B_PipelineNextPushStep - 1].P3 > 0) AND (GVL_1.Step_Cr_B[GVL.B_PipelineNextPushStep].P3 > 0) THEN
						IF (GVL_1.Step_Cr_B[GVL.B_PipelineNextPushStep - 1].P3 > 0) THEN
							//--------------------------------------------
							// Có Blending:
							// quay lại State100 để preload Motion tiếp
							//--------------------------------------------
							GVL.B_RunState := 100;
				
						ELSE
				
							//--------------------------------------------
							// Không Blending:
							// không preload tiếp.
							// Chờ Motion hiện tại Done + Check Position.
							//--------------------------------------------
							//GVL.B_RunState := 120;
							GVL.B_RunState := 100;
				
						END_IF;
					ELSE
						GVL.B_RunState := 120;
					END_IF;
			
			
				ELSIF GVL.B_PushMotionError THEN
			
					GVL.B_PushMotionReq := FALSE;
			
					GVL.B_RunAlarm := TRUE;
					GVL.B_RunAlarmCode := 3001;
					GVL.B_RunErrorStep :=
						GVL.B_PipelineNextPushStep;
			
					GVL.B_RunState := 900;
			
				END_IF;

    120: // WAIT CURRENT STEP DONE
		IF GVL.B_MotionErrorPulse THEN

			GVL.B_RunAlarm := TRUE;
			GVL.B_RunErrorStep := GVL.B_MotionErrorStep;
			GVL.B_RunAlarmCode := GVL.B_MotionErrorCode;
	
			GVL.B_MotionErrorPulse := FALSE;
			GVL.B_RunState := 900;
	
	
		ELSIF GVL.B_MotionDonePulse
			  AND (GVL.B_MotionDoneStep = GVL.B_RunStep)
		THEN
	
			//--------------------------------------------
			// Tiêu thụ Done của step hiện tại
			//--------------------------------------------
			GVL.B_MotionDonePulse := FALSE;
			GVL.B_MotionDoneStep := 0;
	
			//--------------------------------------------
			// Sang step tiếp theo
			//--------------------------------------------
			GVL.B_RunStep :=
				GVL.B_RunStep + 1;
	
			IF (GVL.B_RunStep <= GVL.B_LengthStep)
			   AND F_IsMotionCmd(
					GVL_1.Step_Cr_B[GVL.B_RunStep].Cmd
			   )
			THEN
	
				//----------------------------------------
				// Đồng bộ step tiếp theo cần Push
				//----------------------------------------
// 				GVL.B_PipelineNextPushStep :=
// 					GVL.B_RunStep;
				GVL.B_RunState := 100;
				IF (GVL.B_RunMode = 1) THEN
					GVL.B_StepHold := TRUE;
				END_IF;
				
	
			ELSE
	
				// Gặp END_WHILE hoặc logic khác
				GVL.B_RunState := 130;
	
			END_IF;
	
		END_IF;
		



    130: // WAIT ALL MOTION CLEAR BEFORE LOGIC

		//--------------------------------------------------------
		// Chờ queue và toàn bộ slot motion thực sự sạch
		//--------------------------------------------------------
		IF (GVL.B_MotionCount <= 0)
		   AND (GVL.B_ActiveMotionCount <= 0)
		   AND NOT GVL.B_MotionManagerBusy
		THEN
			//----------------------------------------------------
			// Reset trạng thái phiên pipeline vừa kết thúc
			//----------------------------------------------------
			GVL.B_PipelineActive := FALSE;
// 			GVL.B_PipelineNextPushStep := 0;
// 	
// 			GVL.B_PushMotionReq := FALSE;
// 			GVL.B_PushMotionDone := FALSE;
// 			GVL.B_PushMotionError := FALSE;
// 	
// 			//----------------------------------------------------
// 			// Xóa phản hồi completion của chuỗi motion vừa chạy
// 			//----------------------------------------------------
// 			GVL.B_MotionDonePulse := FALSE;
// 			GVL.B_MotionDoneStep := 0;
// 	
// 			GVL.B_MotionErrorPulse := FALSE;
// 			GVL.B_MotionErrorStep := 0;
// 			GVL.B_MotionErrorCode := 0;
	
			//----------------------------------------------------
			// Quay lại READ STEP để chạy lệnh logic:
			// END_WHILE, IF, WAIT, END...
			//----------------------------------------------------
			GVL.B_RunState := 0;
		END_IF;
		
	140: // WAIT MOTION CLEAR BEFORE WHILE RESTART

		//--------------------------------------------------------
		// Chờ toàn bộ motion của vòng hiện tại hoàn thành
		//--------------------------------------------------------
		IF (GVL.B_MotionCount <= 0)
		   AND (GVL.B_ActiveMotionCount <= 0)
		   AND NOT GVL.B_MotionManagerBusy
		THEN
			//----------------------------------------------------
			// Hạ request của pipeline
			//----------------------------------------------------
			GVL.B_PushMotionReq := FALSE;
			GVL.B_PipelineActive := FALSE;
	
			//----------------------------------------------------
			// Sang bước reset handshake
			//----------------------------------------------------
			MotionCycleResetScan_B := 0;
			GVL.B_RunState := 141;
		END_IF;
		
	141: // RESET MOTION PIPELINE BEFORE NEXT WHILE LOOP

		CASE MotionCycleResetScan_B OF
	
			0:
				//------------------------------------------------
				// Scan thứ nhất: xóa các tín hiệu phiên cũ
				//------------------------------------------------
				GVL.B_PushMotionReq := FALSE;
				GVL.B_PushMotionDone := FALSE;
				GVL.B_PushMotionError := FALSE;
	
				GVL.B_PipelineActive := FALSE;
				GVL.B_PipelineNextPushStep := 0;
	
				GVL.B_MotionDonePulse := FALSE;
				GVL.B_MotionDoneStep := 0;
	
				GVL.B_MotionErrorPulse := FALSE;
				GVL.B_MotionErrorStep := 0;
				GVL.B_MotionErrorCode := 0;
	
				MotionCycleResetScan_B := 1;
	
	
			1:
				//------------------------------------------------
				// Scan thứ hai:
				// fbPushMotion_B đã được gọi với Execute=FALSE.
				// Motion FB đã được gọi với Start=FALSE.
				//------------------------------------------------
				IF NOT GVL.B_PushMotionReq
				   AND (GVL.B_MotionCount <= 0)
				   AND (GVL.B_ActiveMotionCount <= 0)
				   AND NOT GVL.B_MotionManagerBusy
				THEN
					MotionCycleResetScan_B := 0;
	
					//--------------------------------------------
					// Bây giờ mới quay lại WHILE
					//--------------------------------------------
					GVL.B_RunStep := WhileReturnStep_B;
					GVL.B_RunState := 0;
				END_IF;
	
		END_CASE;
	
    900: // ERROR
        GVL.B_RunBusy := FALSE;
        GVL.B_PushMotionReq := FALSE;
        GVL.B_PipelineActive := FALSE;

END_CASE;


//====================================================
// FB Push Motion Queue phải gọi mỗi scan
//====================================================
fbPushMotion_B(
    Execute := GVL.B_PushMotionReq,
    Item := GVL.B_PushMotionItem
);

GVL.B_PushMotionDone  := fbPushMotion_B.Done;
GVL.B_PushMotionError := fbPushMotion_B.Error;
END_ACTION

ACTION PRG_B_MotionManager:
// ACTION/POU: PRG_B_MotionManager
// Create B-specific local FB instances/variables. Do NOT reuse Robot A motion FB instances.
// Required local names can be copied from PRG_A_MotionManager declaration and renamed with _B.


                  
                    
                      //====================================================
// PRG_B_MotionManager
// Controlled Pipeline Motion Manager
// - Chạy nền liên tục.
// - Có queue và slot rảnh thì Pop motion vào slot.
// - Slot Accepted thì hạ Start để FB Motion chạy tiếp.
// - Slot Done thì báo về Interpreter bằng A_MotionDonePulse.
// - Slot Error thì báo lỗi đúng SourceStep.
//====================================================


//====================================================
// ABORT REQUEST
// Ưu tiên cao nhất trong MotionManager
// Dùng khi Stop / Alarm / Reset
//====================================================
IF GVL.B_MotionAbortReq OR GVL.X[7] THEN

    PopReq_B := FALSE;

    GVL.B_MotionHead := 1;
    GVL.B_MotionTail := 1;
    GVL.B_MotionCount := 0;
	GVL.B_PipelineUsedCount := 0;
    FOR i := 1 TO 3 DO
        GVL.B_MoveSlotStart[i] := FALSE;
        GVL.B_MoveSlotBusy[i] := FALSE;

        GVL.B_MoveSlotAccepted[i] := FALSE;
        GVL.B_MoveSlotDone[i] := FALSE;
        GVL.B_MoveSlotError[i] := FALSE;
        GVL.B_MoveSlotErrorID[i] := 0;
		GVL.B_MoveSlotReleasePending[i] := FALSE;
        GVL.B_MoveSlotCmd[i] := E_RobotCmd.CMD_NOP;
		
    END_FOR;

    GVL.B_ActiveMotionCount := 0;

    GVL.B_MotionManagerBusy := FALSE;
    GVL.B_MotionManagerDone := FALSE;
    GVL.B_MotionManagerError := FALSE;
    GVL.B_MotionManagerState := 0;

    GVL.B_MotionDonePulse := FALSE;
    GVL.B_MotionErrorPulse := FALSE;

    GVL.B_MotionAbortReq := FALSE;
    GVL.B_MotionAbortDone := TRUE;

ELSE

	// Luôn gọi FB MoveP/L/C mỗi scan
	
	CASE GVL.B_MotionManagerState OF
	
		0: // IDLE / READY
	
			GVL.B_MotionManagerDone := FALSE;
	
			// Nếu có motion trong queue và còn slot rảnh thì lấy ra chạy
			IF (GVL.B_MotionCount > 0) AND (F_GetFreeMoveSlot_B() > 0) THEN
				GVL.B_MotionManagerBusy := TRUE;
				PopReq_B := TRUE;
	
				GVL.B_MotionManagerState := 10;
	
			ELSE
				// Không còn queue và không còn slot active
				IF GVL.B_ActiveMotionCount <= 0 THEN
					GVL.B_MotionManagerBusy := FALSE;
				END_IF;
			END_IF;
	
	
		10: // WAIT POP DONE
	
			IF fbPop_B.Done THEN
				PopReq_B := FALSE;
	
				item_PRG_B_MotionManager := fbPop_B.Item;
				freeSlot_B := F_GetFreeMoveSlot_B();
	
				IF freeSlot_B > 0 THEN
	
					// Gán item vào slot rảnh
					GVL.B_MoveSlotItem[freeSlot_B] := item_PRG_B_MotionManager;
					GVL.B_MoveSlotCmd[freeSlot_B]  := item_PRG_B_MotionManager.Cmd;
	
					// Reset trạng thái slot trước khi Start
					GVL.B_MoveSlotBusy[freeSlot_B]     := TRUE;
					GVL.B_MoveSlotStart[freeSlot_B]    := TRUE;
					GVL.B_MoveSlotAccepted[freeSlot_B] := FALSE;
					GVL.B_MoveSlotDone[freeSlot_B]     := FALSE;
					GVL.B_MoveSlotError[freeSlot_B]    := FALSE;
					
					GVL.B_MoveSlotErrorID[freeSlot_B] := 0;

					GVL.B_MoveSlotReleasePending[freeSlot_B] := FALSE;
					
					// Ghi nhớ chính xác slot vừa cấp
   					WaitAcceptSlot_B := freeSlot_B;
	
					// Tăng số motion đang active
					//GVL.B_ActiveMotionCount := GVL.B_ActiveMotionCount + 1;
	
					GVL.B_MotionManagerState := 20;
	
				ELSE
					// Trường hợp hiếm: vừa Pop xong nhưng slot không còn rảnh
					GVL.B_MotionManagerState := 30;
				END_IF;
			END_IF;
	
			IF fbPop_B.Empty THEN
				PopReq_B := FALSE;
				GVL.B_MotionManagerState := 30;
			END_IF;
	
	
		20: // WAIT COMMAND ACCEPTED
			
		//--------------------------------------------------------
			// Chỉ chờ đúng slot vừa được State 10 cấp lệnh
			//--------------------------------------------------------
			IF (WaitAcceptSlot_B >= 1)
			   AND (WaitAcceptSlot_B <= 3)
			THEN
		
				//----------------------------------------------------
				// Slot vẫn phải thuộc quyền sở hữu của Manager
				//----------------------------------------------------
				IF GVL.B_MoveSlotBusy[WaitAcceptSlot_B] THEN
		
					//------------------------------------------------
					// Lệnh đã được FB Move nhận
					//------------------------------------------------
					IF GVL.B_MoveSlotAccepted[WaitAcceptSlot_B] THEN
		
						GVL.B_MoveSlotStart[WaitAcceptSlot_B] := FALSE;
		
						// Đã hoàn thành handshake Accepted
						WaitAcceptSlot_B := 0;
		
						//--------------------------------------------
						// PipelineLength = 1:
						// Không Pop thêm khi còn motion đang chạy.
						// Sang State 30 chờ motion hoàn thành.
						//--------------------------------------------
						GVL.B_MotionManagerState := 30;
		
		
					ELSIF GVL.B_MoveSlotError[WaitAcceptSlot_B] THEN
		
						GVL.B_MotionManagerError := TRUE;
		
						GVL.B_MotionErrorPulse := TRUE;
						GVL.B_MotionErrorStep :=
							GVL.B_MoveSlotItem[WaitAcceptSlot_B].SourceStep;
		
						GVL.B_MotionErrorCode :=
							GVL.B_MoveSlotErrorID[WaitAcceptSlot_B];
		
						WaitAcceptSlot_B := 0;
		
						GVL.B_MotionManagerState := 900;
		
					END_IF;
		
				END_IF;
		
			ELSE
		
				//----------------------------------------------------
				// Không có slot nào đang chờ Accepted.
				// Đây là trạng thái bất thường, quay về quản lý queue.
				//----------------------------------------------------
				GVL.B_MotionManagerState := 30;
		
			END_IF;
	
		30: // WAIT / CONTINUE PIPELINE
	
			// Nếu sau đó Interpreter push thêm queue và có slot rảnh thì tiếp tục chạy
			IF (GVL.B_MotionCount > 0) AND (F_GetFreeMoveSlot_B() > 0) THEN
				GVL.B_MotionManagerBusy := TRUE;
				PopReq_B := TRUE;
				GVL.B_MotionManagerState := 10;
	
			// Nếu không còn queue và không còn motion active thì MotionManager rảnh
			ELSIF (GVL.B_MotionCount <= 0) AND (GVL.B_ActiveMotionCount <= 0) THEN
				GVL.B_MotionManagerBusy := FALSE;
				GVL.B_MotionManagerDone := TRUE;
				GVL.B_MotionManagerState := 0;
			END_IF;
	
	
		900: // ERROR
	
			PopReq_B := FALSE;
	
			// Dừng cấp thêm motion mới
			FOR i := 1 TO 3 DO
				GVL.B_MoveSlotStart[i] := FALSE;
			END_FOR;
	
			GVL.B_MotionManagerBusy := FALSE;
			GVL.B_MotionManagerError := TRUE;
	
			GVL.B_MotionManagerState := 0;
	
	END_CASE;
END_IF;
//====================================================
// Gọi FB Pop mỗi scan
//====================================================
fbPop_B(
    Execute := PopReq_B
);



//============================================================
// CALL MOTION SLOT FB
// Tất cả FB phải được gọi liên tục mỗi scan.
//
// Khi slot không sử dụng hoặc không đúng loại lệnh:
// Start của FB tương ứng phải bằng FALSE.
// Nhờ vậy LastStart và State bên trong FB được cập nhật đúng.
//============================================================

FOR i := 1 TO 3 DO

    //--------------------------------------------------------
    // Chuẩn bị tọa độ
    //--------------------------------------------------------
    IF GVL.B_MoveSlotBusy[i] THEN

        CASE GVL.B_MoveSlotCmd[i] OF

            E_RobotCmd.CMD_MovP,
            E_RobotCmd.CMD_MovL:

//                 SlotPos_B[i] :=
//                     F_GetPointSMC_B(
//                         GVL.B_MoveSlotItem[i].PointNo
//                     );
				IF GVL.B_MoveSlotItem[i].UseDirectPosition THEN
					SlotPos_B[i].c.X := GVL.B_MoveSlotItem[i].DirectPosition.X;
					SlotPos_B[i].c.Y := GVL.B_MoveSlotItem[i].DirectPosition.Y;
					SlotPos_B[i].c.Z := GVL.B_MoveSlotItem[i].DirectPosition.Z;
					SlotPos_B[i].c.A := GVL.B_MoveSlotItem[i].DirectPosition.A;
				ELSE
					SlotPos_B[i] := F_GetPointSMC_B(GVL.B_MoveSlotItem[i].PointNo);
				END_IF;



            E_RobotCmd.CMD_MovC:

                SlotMidPos_B[i] :=
                    F_GetPointSMC_B(
                        GVL.B_MoveSlotItem[i].MidPointNo
                    );

                SlotEndPos_B[i] :=
                    F_GetPointSMC_B(
                        GVL.B_MoveSlotItem[i].EndPointNo
                    );

        END_CASE;

    END_IF;


    //--------------------------------------------------------
    // MoveP
    // Luôn gọi mỗi scan
    //--------------------------------------------------------
    fbMoveP_B[i](
        Start :=
            GVL.B_MoveSlotBusy[i]
            AND
            (GVL.B_MoveSlotCmd[i] = E_RobotCmd.CMD_MovP)
            AND
            GVL.B_MoveSlotStart[i],
		Release := GVL.B_MoveSlotReleasePending[i],
        AxisGroup := SCARA_B,
        Item := GVL.B_MoveSlotItem[i],
        PositionIn := SlotPos_B[i],
        //CoordSystem := GVL.RB_B.COORD
		CoordSystem := SEL(
			GVL.B_MoveSlotItem[i].UseDirectPosition,
			//GVL.RB_B.COORD,
			SMC_COORD_SYSTEM.MCS,
			GVL.B_MoveSlotItem[i].DirectCoordSystem)

    );


    //--------------------------------------------------------
    // MoveL
    // Luôn gọi mỗi scan
    //--------------------------------------------------------
    fbMoveL_B[i](
        Start :=
            GVL.B_MoveSlotBusy[i]
            AND
            (GVL.B_MoveSlotCmd[i] = E_RobotCmd.CMD_MovL)
            AND
            GVL.B_MoveSlotStart[i],

        AxisGroup := SCARA_B,
        Item := GVL.B_MoveSlotItem[i],
        PositionIn := SlotPos_B[i],
        //CoordSystem := GVL.RB_B.COORD
		CoordSystem := SEL(
			GVL.B_MoveSlotItem[i].UseDirectPosition,
			//GVL.RB_B.COORD,
			SMC_COORD_SYSTEM.MCS,
			GVL.B_MoveSlotItem[i].DirectCoordSystem)

    );


    //--------------------------------------------------------
    // MoveC
    // Luôn gọi mỗi scan
    //--------------------------------------------------------
    fbMoveC_B[i](
        Start :=
            GVL.B_MoveSlotBusy[i]
            AND
            (GVL.B_MoveSlotCmd[i] = E_RobotCmd.CMD_MovC)
            AND
            GVL.B_MoveSlotStart[i],

        AxisGroup := SCARA_B,
        Item := GVL.B_MoveSlotItem[i],
        MidPosition := SlotMidPos_B[i],
        EndPosition := SlotEndPos_B[i],
        //CoordSystem := GVL.RB_B.COORD
		CoordSystem := SMC_COORD_SYSTEM.MCS
    );


	



    //--------------------------------------------------------
    // Chọn trạng thái trả về theo loại lệnh của slot
    //--------------------------------------------------------
    IF GVL.B_MoveSlotBusy[i] THEN

        CASE GVL.B_MoveSlotCmd[i] OF

            //================================================
            // MOVP
            //================================================
            E_RobotCmd.CMD_MovP:

                GVL.B_MoveSlotAccepted[i] :=
                    fbMoveP_B[i].Accepted;

                GVL.B_MoveSlotDone[i] :=
                    fbMoveP_B[i].Done;

                GVL.B_MoveSlotError[i] :=
                    fbMoveP_B[i].Error;

                GVL.B_MoveSlotErrorID[i] :=
                    fbMoveP_B[i].ErrorID_Custom;


            //================================================
            // MOVL
            //================================================
            E_RobotCmd.CMD_MovL:

                GVL.B_MoveSlotAccepted[i] :=
                    fbMoveL_B[i].Accepted;

                GVL.B_MoveSlotDone[i] :=
                    fbMoveL_B[i].Done;

                GVL.B_MoveSlotError[i] :=
                    fbMoveL_B[i].Error;

                GVL.B_MoveSlotErrorID[i] :=
                    fbMoveL_B[i].ErrorID_Custom;


            //================================================
            // MOVC
            //================================================
            E_RobotCmd.CMD_MovC:

                GVL.B_MoveSlotAccepted[i] :=
                    fbMoveC_B[i].Accepted;

                GVL.B_MoveSlotDone[i] :=
                    fbMoveC_B[i].Done;

                GVL.B_MoveSlotError[i] :=
                    fbMoveC_B[i].Error;

                GVL.B_MoveSlotErrorID[i] :=
                    fbMoveC_B[i].ErrorID_Custom;

        END_CASE;

    END_IF;

END_FOR;


//------------------------------------------------------------
// GLOBAL MOTION ERROR MONITOR
//
// Kiểm tra tất cả Move Slot mỗi scan.
// Giữ nguyên cơ chế MotionErrorPulse cũ để báo Interpreter.
//------------------------------------------------------------
IF NOT GVL.B_MotionErrorPulse THEN

    FOR i := 1 TO 3 DO

        IF GVL.B_MoveSlotBusy[i] AND GVL.B_MoveSlotError[i]
        THEN

            //--------------------------------------------
            // MotionManager có lỗi
            //--------------------------------------------
            GVL.B_MotionManagerError := TRUE;

            //--------------------------------------------
            // Xung báo Interpreter
            //--------------------------------------------
            GVL.B_MotionErrorPulse := TRUE;

            //--------------------------------------------
            // Step gây lỗi
            //--------------------------------------------
            GVL.B_MotionErrorStep := GVL.B_MoveSlotItem[i].SourceStep;

            //--------------------------------------------
            // Error Code của FB
            //--------------------------------------------
            GVL.B_MotionErrorCode := GVL.B_MoveSlotErrorID[i];

            //--------------------------------------------
            // Có thể lưu thêm Slot để debug
            //--------------------------------------------
            GVL.B_MotionErrorSlot := i;

            //--------------------------------------------
            // Manager chuyển ERROR
            //--------------------------------------------
            GVL.B_MotionManagerState := 900;

            EXIT;

        END_IF;

    END_FOR;

END_IF;

// RELEASE SLOT WHEN DONE
FOR i := 1 TO 3 DO

    IF GVL.B_MoveSlotBusy[i]
       AND GVL.B_MoveSlotDone[i]
    THEN

        // Báo Interpreter
        GVL.B_MotionDoneStep :=
            GVL.B_MoveSlotItem[i].SourceStep;

        GVL.B_MotionDonePulse := TRUE;

        // Release slot
        GVL.B_MoveSlotStart[i] := FALSE;
        GVL.B_MoveSlotBusy[i] := FALSE;
        GVL.B_MoveSlotAccepted[i] := FALSE;
        GVL.B_MoveSlotDone[i] := FALSE;
        GVL.B_MoveSlotError[i] := FALSE;
        GVL.B_MoveSlotErrorID[i] := 0;

        GVL.B_MoveSlotCmd[i] :=
            E_RobotCmd.CMD_NOP;
		GVL.B_MoveSlotReleasePending[i] := TRUE; // Set release = TRUE
		
		//------------------------------------------------
		// Motion đã thực sự rời pipeline
		//------------------------------------------------
		IF GVL.B_PipelineUsedCount > 0 THEN
			GVL.B_PipelineUsedCount :=
				GVL.B_PipelineUsedCount - 1;
		END_IF;
	
    END_IF;
END_FOR;

//============================================================
// RECALCULATE ACTIVE MOTION COUNT
//
// A_ActiveMotionCount luôn phản ánh đúng số slot Busy,
// không phụ thuộc việc cộng/trừ có bị bỏ sót hay không.
//============================================================
ActiveCountCalc := 0;

FOR i := 1 TO 3 DO

    IF GVL.B_MoveSlotBusy[i] THEN
        ActiveCountCalc := ActiveCountCalc + 1;
    END_IF;

END_FOR;

GVL.B_ActiveMotionCount := ActiveCountCalc;




//====================================================
// FINALIZE MOTION MANAGER
// Chỉ kết thúc khi Manager đã vào trạng thái WAIT
// Không được reset State 10/20 khi vừa Pop lệnh.
//====================================================
IF (GVL.B_MotionManagerState = 30)
   AND (GVL.B_MotionCount <= 0)
   AND (GVL.B_ActiveMotionCount <= 0)
THEN

    GVL.B_MotionManagerBusy := FALSE;
    GVL.B_MotionManagerDone := TRUE;
    GVL.B_MotionManagerState := 0;

END_IF;
END_ACTION

ACTION _Main_Process_Test:
// PROCESS 
IF Ena_Test THEN
	GVL.RB_A.COORD := 1;
	GVL.RB_B.COORD := 1;
	IF NOT Just_Start_Test THEN
		A_Test_Motion_Run := FALSE;
		B_Test_Motion_Run := FALSE;
		Process_B_Test := 0;
		Process_A_Test := 0;
	END_IF
	Just_Start_Test := TRUE;
	A_Test_Motion_Run := TRUE;
	A_Test_Motion();
	B_Test_Motion_Run := TRUE;
	B1_Test_Motion();

ELSIF NOT Ena_Test THEN

	A_Test_Motion_Run := FALSE;
	B_Test_Motion_Run := FALSE;
	Process_B_Test := 0;
	Process_A_Test := 0;
END_IF	 
{endregion}
END_ACTION

